C09078=1071.190,436.520,-116.526,176.537,35.842,156.699
C09079=1071.199,436.766,-116.574,176.544,35.855,156.702
C09080=1071.208,437.011,-116.622,176.552,35.868,156.705
C09081=1071.216,437.256,-116.669,176.561,35.881,156.709
C09082=1071.225,437.501,-116.716,176.568,35.894,156.712
C09083=1071.234,437.746,-116.764,176.576,35.908,156.716
C09084=1071.243,437.991,-116.811,176.585,35.921,156.719
C09085=1071.251,438.238,-116.859,176.593,35.934,156.722
C09086=1071.260,438.482,-116.906,176.600,35.947,156.726
C09087=1071.269,438.727,-116.954,176.609,35.961,156.729
C09088=1071.279,438.973,-117.001,176.617,35.974,156.733
C09089=1071.287,439.218,-117.049,176.626,35.988,156.736
C09090=1071.296,439.463,-117.097,176.633,36.001,156.739
C09091=1071.304,439.709,-117.145,176.641,36.015,156.743
C09092=1071.313,439.954,-117.193,176.650,36.029,156.747
C09093=1071.322,440.198,-117.241,176.658,36.042,156.750
C09094=1071.331,440.444,-117.289,176.667,36.056,156.754
C09095=1071.340,440.689,-117.337,176.675,36.069,156.757
C09096=1071.348,440.933,-117.385,176.684,36.083,156.761
C09097=1071.358,441.193,-117.437,176.693,36.098,156.764
C09098=1071.367,441.451,-117.487,176.702,36.113,156.768
C09099=1071.376,441.709,-117.538,176.711,36.127,156.772
C09100=1071.386,441.968,-117.589,176.720,36.142,156.776
C09101=1071.395,442.213,-117.637,176.728,36.156,156.779
C09102=1071.404,442.459,-117.686,176.737,36.170,156.783
C09103=1071.413,442.703,-117.734,176.745,36.184,156.787
C09104=1071.422,442.949,-117.782,176.754,36.199,156.791
C09105=1071.431,443.193,-117.831,176.763,36.213,156.794
C09106=1071.440,443.438,-117.880,176.771,36.227,156.798
C09107=1071.449,443.684,-117.929,176.780,36.241,156.802
C09108=1071.458,443.928,-117.977,176.789,36.256,156.805
C09109=1071.467,444.173,-118.026,176.798,36.270,156.809
C09110=1071.476,444.418,-118.075,176.806,36.285,156.813
C09111=1071.485,444.663,-118.123,176.816,36.299,156.817
C09112=1071.494,444.908,-118.172,176.825,36.314,156.821
C09113=1071.503,445.153,-118.222,176.834,36.329,156.824
C09114=1071.512,445.399,-118.271,176.842,36.343,156.828
C09115=1071.522,445.642,-118.320,176.851,36.358,156.832
C09116=1071.531,445.887,-118.369,176.861,36.373,156.836
C09117=1071.540,446.133,-118.418,176.870,36.388,156.840
C09118=1071.549,446.377,-118.468,176.879,36.402,156.844
C09119=1071.559,446.622,-118.516,176.888,36.417,156.848
C09120=1071.568,446.868,-118.565,176.898,36.433,156.852
C09121=1071.577,447.112,-118.615,176.907,36.447,156.856
C09122=1071.586,447.356,-118.665,176.916,36.463,156.860
C09123=1071.596,447.601,-118.713,176.926,36.477,156.864
C09124=1071.606,447.847,-118.763,176.934,36.493,156.868
C09125=1071.615,448.091,-118.813,176.943,36.508,156.872
C09126=1071.624,448.334,-118.862,176.952,36.523,156.876
C09127=1071.634,448.579,-118.911,176.959,36.538,156.880
C09128=1071.646,448.822,-118.959,176.967,36.552,156.883
C09129=1071.658,449.067,-119.006,176.976,36.566,156.887
C09130=1071.672,449.312,-119.053,176.983,36.579,156.891
C09131=1071.687,449.558,-119.100,176.990,36.592,156.894
C09132=1071.704,449.803,-119.144,176.997,36.604,156.897
C09133=1071.353,449.802,-119.394,176.982,36.746,156.935
C09134=1071.337,449.558,-119.348,176.975,36.734,156.932
C09135=1071.322,449.311,-119.302,176.968,36.722,156.929
C09136=1071.308,449.066,-119.255,176.960,36.708,156.925
C09137=1071.295,448.822,-119.208,176.953,36.695,156.921
C09138=1071.283,448.577,-119.160,176.944,36.680,156.918
C09139=1071.272,448.333,-119.111,176.936,36.666,156.914
C09140=1071.264,448.089,-119.062,176.927,36.650,156.910
C09141=1071.254,447.846,-119.012,176.918,36.636,156.906
C09142=1071.245,447.601,-118.962,176.908,36.620,156.902
C09143=1071.236,447.356,-118.913,176.899,36.605,156.898
C09144=1071.225,447.112,-118.864,176.890,36.590,156.894
C09145=1071.216,446.867,-118.814,176.880,36.575,156.890
C09146=1071.207,446.622,-118.765,176.871,36.560,156.886
C09147=1071.198,446.377,-118.715,176.862,36.545,156.882
C09148=1071.188,446.132,-118.667,176.853,36.531,156.878
C09149=1071.179,445.888,-118.617,176.844,36.516,156.874
C09150=1071.170,445.642,-118.568,176.834,36.501,156.870
C09151=1071.161,445.397,-118.519,176.825,36.486,156.866
C09152=1071.151,445.153,-118.470,176.816,36.472,156.862
C09153=1071.142,444.908,-118.421,176.806,36.457,156.858
C09154=1071.133,444.663,-118.371,176.798,36.443,156.855
C09155=1071.124,444.418,-118.322,176.789,36.428,156.851
C09156=1071.115,444.173,-118.274,176.780,36.413,156.847
C09157=1071.106,443.928,-118.225,176.771,36.399,156.843
C09158=1071.097,443.683,-118.176,176.762,36.385,156.839
C09159=1071.088,443.438,-118.128,176.753,36.370,156.836
C09160=1071.079,443.193,-118.079,176.744,36.356,156.832
C09161=1071.069,442.948,-118.030,176.735,36.342,156.828
C09162=1071.061,442.706,-117.982,176.727,36.328,156.825
C09163=1071.052,442.463,-117.933,176.718,36.314,156.821
C09164=1071.042,442.220,-117.885,176.710,36.300,156.817
C09165=1071.034,441.978,-117.838,176.701,36.286,156.814
C09166=1071.025,441.735,-117.790,176.693,36.272,156.810
C09167=1071.016,441.493,-117.742,176.684,36.259,156.806
C09168=1071.007,441.250,-117.694,176.676,36.245,156.803
C09169=1070.999,441.007,-117.647,176.667,36.231,156.799
C09170=1070.989,440.762,-117.598,176.659,36.217,156.796
C09171=1070.981,440.517,-117.550,176.650,36.203,156.792
C09172=1070.971,440.272,-117.502,176.642,36.190,156.789
C09173=1070.962,440.027,-117.454,176.633,36.176,156.785
C09174=1070.954,439.782,-117.406,176.625,36.163,156.782
C09175=1070.945,439.537,-117.358,176.616,36.149,156.778
C09176=1070.937,439.291,-117.310,176.608,36.135,156.774
C09177=1070.928,439.046,-117.263,176.599,36.122,156.771
C09178=1070.918,438.801,-117.215,176.591,36.108,156.768
C09179=1070.910,438.556,-117.167,176.584,36.095,156.764
C09180=1070.901,438.311,-117.120,176.575,36.082,156.761
C09181=1070.892,438.065,-117.072,176.567,36.068,156.757
C09182=1070.883,437.820,-117.024,176.559,36.055,156.754
C09183=1070.874,437.575,-116.977,176.550,36.042,156.750
C09184=1070.866,437.330,-116.929,176.543,36.029,156.747
C09185=1070.857,437.085,-116.881,176.535,36.016,156.744
C09186=1070.848,436.839,-116.834,176.526,36.003,156.741
C09187=1070.839,436.594,-116.787,176.518,35.990,156.737
C09188=1070.831,436.349,-116.740,176.511,35.977,156.734
C09189=1070.822,436.104,-116.693,176.502,35.964,156.731
C09190=1070.813,435.859,-116.645,176.494,35.951,156.727
C09191=1070.805,435.612,-116.597,176.486,35.938,156.724
C09192=1070.796,435.367,-116.550,176.479,35.925,156.721
C09193=1070.787,435.122,-116.503,176.471,35.912,156.717
C09194=1070.779,434.876,-116.457,176.463,35.900,156.714
C09195=1070.770,434.632,-116.409,176.455,35.887,156.711
C09196=1070.761,434.386,-116.362,176.447,35.874,156.708
C09197=1070.753,434.140,-116.316,176.440,35.862,156.705
C09198=1070.744,433.895,-116.269,176.432,35.849,156.701
C09199=1070.736,433.651,-116.222,176.424,35.837,156.698
C09200=1070.727,433.405,-116.175,176.417,35.824,156.695
C09201=1070.719,433.160,-116.128,176.409,35.811,156.692
C09202=1070.711,432.914,-116.081,176.402,35.799,156.689
C09203=1070.702,432.668,-116.034,176.394,35.787,156.686
C09204=1070.694,432.423,-115.988,176.387,35.774,156.683
C09205=1070.685,432.177,-115.941,176.379,35.762,156.679
C09206=1070.677,431.933,-115.895,176.372,35.750,156.676
C09207=1070.669,431.686,-115.849,176.364,35.738,156.673
C09208=1070.661,431.441,-115.802,176.357,35.725,156.670
C09209=1070.652,431.195,-115.755,176.349,35.713,156.667
C09210=1070.643,430.950,-115.709,176.342,35.701,156.664
C09211=1070.635,430.705,-115.663,176.334,35.689,156.661
C09212=1070.627,430.459,-115.617,176.327,35.677,156.658
C09213=1070.618,430.213,-115.571,176.320,35.665,156.655
C09214=1070.610,429.968,-115.524,176.312,35.653,156.652
C09215=1070.601,429.723,-115.479,176.305,35.641,156.649
C09216=1070.593,429.477,-115.432,176.297,35.629,156.646
C09217=1070.585,429.231,-115.386,176.290,35.617,156.643
C09218=1070.577,428.986,-115.340,176.283,35.606,156.640
C09219=1070.568,428.740,-115.294,176.276,35.594,156.637
C09220=1070.560,428.495,-115.249,176.269,35.582,156.634
C09221=1070.552,428.249,-115.202,176.262,35.570,156.632
C09222=1070.542,427.953,-115.146,176.253,35.556,156.628
C09223=1070.532,427.658,-115.091,176.244,35.542,156.625
C09224=1070.522,427.362,-115.037,176.236,35.528,156.621
C09225=1070.512,427.066,-114.982,176.227,35.514,156.618
C09226=1070.504,426.820,-114.936,176.220,35.503,156.615
C09227=1070.496,426.575,-114.891,176.214,35.492,156.612
C09228=1070.487,426.329,-114.845,176.207,35.480,156.609
C09229=1070.479,426.084,-114.800,176.199,35.469,156.607
C09230=1070.471,425.838,-114.754,176.192,35.457,156.604
C09231=1070.462,425.593,-114.709,176.186,35.446,156.601
C09232=1070.454,425.347,-114.663,176.179,35.435,156.598
C09233=1070.446,425.101,-114.619,176.171,35.423,156.595
C09234=1070.438,424.855,-114.573,176.165,35.412,156.593
C09235=1070.429,424.610,-114.528,176.158,35.401,156.590
C09236=1070.422,424.363,-114.483,176.151,35.390,156.587
C09237=1070.413,424.118,-114.437,176.145,35.379,156.584
C09238=1070.405,423.872,-114.392,176.138,35.368,156.582
C09239=1070.397,423.626,-114.347,176.131,35.357,156.579
C09240=1070.389,423.381,-114.302,176.124,35.346,156.576
C09241=1070.381,423.135,-114.257,176.117,35.335,156.574
C09242=1070.373,422.889,-114.212,176.111,35.324,156.571
C09243=1070.365,422.643,-114.167,176.104,35.313,156.568
C09244=1070.357,422.398,-114.123,176.098,35.302,156.566
C09245=1070.349,422.152,-114.077,176.091,35.291,156.563
C09246=1070.341,421.906,-114.032,176.085,35.280,156.560
C09247=1070.333,421.660,-113.988,176.077,35.269,156.558
C09248=1070.325,421.415,-113.942,176.071,35.259,156.555
C09249=1070.317,421.169,-113.898,176.064,35.248,156.552
C09250=1070.309,420.923,-113.854,176.058,35.237,156.550
C09251=1070.301,420.676,-113.808,176.051,35.227,156.547
C09252=1070.293,420.431,-113.764,176.045,35.216,156.545
C09253=1070.285,420.185,-113.720,176.039,35.205,156.542
C09254=1070.277,419.939,-113.675,176.032,35.195,156.540
C09255=1070.269,419.693,-113.631,176.026,35.184,156.537
C09256=1070.262,419.447,-113.586,176.019,35.174,156.534
C09257=1070.254,419.202,-113.542,176.013,35.164,156.532
C09258=1070.246,418.955,-113.498,176.006,35.153,156.529
C09259=1070.238,418.709,-113.454,176.000,35.143,156.527
C09260=1070.230,418.464,-113.409,175.994,35.132,156.525
C09261=1070.222,418.218,-113.365,175.987,35.122,156.522
C09262=1070.214,417.972,-113.321,175.981,35.112,156.520
C09263=1070.206,417.726,-113.277,175.975,35.101,156.517
C09264=1070.198,417.480,-113.232,175.968,35.091,156.515
C09265=1070.191,417.233,-113.189,175.962,35.081,156.512
C09266=1070.183,416.988,-113.144,175.956,35.071,156.510
C09267=1070.175,416.742,-113.100,175.950,35.061,156.507
C09268=1070.167,416.496,-113.056,175.944,35.050,156.505
C09269=1070.159,416.250,-113.012,175.938,35.040,156.502
C09270=1070.151,416.004,-112.968,175.932,35.030,156.500
C09271=1070.143,415.757,-112.925,175.925,35.020,156.498
C09272=1070.136,415.512,-112.881,175.919,35.010,156.495
C09273=1070.128,415.266,-112.837,175.913,35.000,156.493
C09274=1070.120,415.020,-112.793,175.907,34.990,156.490
C09275=1070.112,414.774,-112.749,175.901,34.980,156.488
C09276=1070.104,414.527,-112.706,175.894,34.970,156.486
C09277=1070.097,414.281,-112.662,175.889,34.960,156.483
C09278=1070.088,414.004,-112.613,175.882,34.949,156.481
C09279=1070.079,413.728,-112.564,175.875,34.938,156.478
C09280=1070.071,413.451,-112.515,175.869,34.927,156.475
C09281=1070.061,413.174,-112.466,175.862,34.916,156.473
C09282=1070.050,412.806,-112.402,175.853,34.902,156.469
C09283=1070.039,412.438,-112.336,175.843,34.887,156.466
C09284=1070.027,412.069,-112.272,175.835,34.873,156.463
C09285=1070.015,411.700,-112.207,175.826,34.859,156.459
C09286=1070.007,411.454,-112.164,175.820,34.849,156.457
C09287=1070.000,411.208,-112.121,175.815,34.840,156.455
C09288=1069.992,410.962,-112.077,175.809,34.830,156.452
C09289=1069.984,410.715,-112.035,175.803,34.821,156.450
C09290=1069.977,410.470,-111.991,175.797,34.811,156.448
C09291=1069.969,410.224,-111.948,175.791,34.802,156.446
C09292=1069.962,409.977,-111.906,175.786,34.793,156.444
C09293=1069.954,409.731,-111.862,175.780,34.783,156.441
C09294=1069.946,409.485,-111.820,175.774,34.774,156.439
C09295=1069.939,409.239,-111.777,175.769,34.764,156.437
C09296=1069.932,408.993,-111.733,175.763,34.755,156.435
C09297=1069.923,408.746,-111.691,175.757,34.746,156.433
C09298=1069.916,408.501,-111.648,175.751,34.737,156.431
C09299=1069.909,408.254,-111.605,175.746,34.727,156.428
C09300=1069.901,408.008,-111.563,175.740,34.718,156.426
C09301=1069.894,407.762,-111.520,175.734,34.709,156.424
C09302=1069.887,407.515,-111.477,175.729,34.700,156.422
C09303=1069.879,407.269,-111.435,175.723,34.690,156.420
C09304=1069.871,407.023,-111.391,175.717,34.681,156.418
C09305=1069.864,406.776,-111.349,175.712,34.672,156.416
C09306=1069.857,406.530,-111.307,175.707,34.663,156.413
C09307=1069.849,406.283,-111.264,175.701,34.654,156.411
C09308=1069.842,406.038,-111.222,175.696,34.645,156.409
C09309=1069.835,405.792,-111.179,175.690,34.636,156.407
C09310=1069.826,405.545,-111.136,175.684,34.627,156.405
C09311=1069.819,405.299,-111.094,175.679,34.618,156.403
C09312=1069.812,405.053,-111.052,175.673,34.609,156.401
C09313=1069.804,404.807,-111.010,175.667,34.600,156.399
C09314=1069.797,404.560,-110.967,175.663,34.592,156.397
C09315=1069.789,404.314,-110.925,175.657,34.583,156.395
C09316=1069.782,404.068,-110.882,175.651,34.574,156.393
C09317=1069.775,403.821,-110.841,175.646,34.565,156.391
C09318=1069.767,403.574,-110.799,175.640,34.557,156.389
C09319=1069.760,403.328,-110.756,175.636,34.548,156.387
C09320=1069.752,403.082,-110.714,175.630,34.539,156.385
C09321=1069.745,402.836,-110.672,175.624,34.530,156.383
C09322=1069.738,402.590,-110.631,175.619,34.522,156.381
C09323=1069.731,402.343,-110.589,175.613,34.513,156.379
C09324=1069.723,402.097,-110.546,175.609,34.505,156.377
C09325=1069.715,401.850,-110.505,175.603,34.496,156.375
C09326=1069.708,401.604,-110.463,175.598,34.487,156.373
C09327=1069.700,401.358,-110.421,175.592,34.479,156.371
C09328=1069.693,401.111,-110.379,175.587,34.470,156.369
C09329=1069.686,400.865,-110.338,175.582,34.462,156.367
C09330=1069.674,400.468,-110.271,175.573,34.448,156.364
C09331=1069.662,400.071,-110.203,175.565,34.434,156.361
C09332=1069.650,399.674,-110.137,175.556,34.421,156.358
C09333=1069.639,399.277,-110.069,175.548,34.408,156.354
C09334=1069.631,399.031,-110.028,175.543,34.399,156.353
C09335=1069.624,398.784,-109.987,175.537,34.391,156.351
C09336=1069.616,398.538,-109.945,175.533,34.383,156.349
C09337=1069.609,398.291,-109.904,175.527,34.374,156.347
C09338=1069.602,398.045,-109.862,175.523,34.366,156.345
C09339=1069.595,397.798,-109.821,175.517,34.358,156.343
C09340=1069.587,397.552,-109.780,175.512,34.350,156.341
C09341=1069.580,397.306,-109.738,175.507,34.341,156.339
C09342=1069.572,397.059,-109.697,175.502,34.333,156.337
C09343=1069.566,396.813,-109.656,175.497,34.325,156.336
C09344=1069.558,396.567,-109.615,175.492,34.317,156.334
C09345=1069.551,396.320,-109.573,175.487,34.309,156.332
C09346=1069.544,396.073,-109.532,175.482,34.301,156.330
C09347=1069.537,395.827,-109.491,175.477,34.293,156.328
C09348=1069.529,395.580,-109.450,175.471,34.284,156.326
C09349=1069.523,395.334,-109.409,175.467,34.277,156.325
C09350=1069.515,395.088,-109.368,175.461,34.268,156.323
C09351=1069.508,394.841,-109.328,175.457,34.261,156.321
C09352=1069.500,394.594,-109.287,175.451,34.253,156.319
C09353=1069.494,394.348,-109.246,175.447,34.245,156.317
C09354=1069.486,394.102,-109.204,175.441,34.237,156.316
C09355=1069.479,393.855,-109.163,175.437,34.229,156.314
C09356=1069.473,393.609,-109.123,175.432,34.221,156.312
C09357=1069.465,393.362,-109.082,175.426,34.213,156.310
C09358=1069.457,393.116,-109.041,175.422,34.205,156.309
C09359=1069.451,392.869,-109.001,175.416,34.197,156.307
C09360=1069.443,392.623,-108.960,175.412,34.190,156.305
C09361=1069.436,392.376,-108.919,175.406,34.182,156.303
C09362=1069.429,392.130,-108.879,175.402,34.174,156.302
C09363=1069.422,391.883,-108.838,175.397,34.166,156.300
C09364=1069.414,391.636,-108.798,175.392,34.159,156.298
C09365=1069.408,391.390,-108.757,175.387,34.151,156.296
C09366=1069.401,391.143,-108.716,175.382,34.143,156.295
C09367=1069.393,390.898,-108.676,175.377,34.136,156.293
C09368=1069.386,390.650,-108.636,175.373,34.128,156.291
C09369=1069.379,390.405,-108.595,175.367,34.120,156.289
C09370=1069.372,390.158,-108.555,175.363,34.113,156.288
C09371=1069.364,389.911,-108.515,175.359,34.105,156.286
C09372=1069.357,389.665,-108.474,175.353,34.098,156.285
C09373=1069.350,389.418,-108.434,175.349,34.090,156.283
C09374=1069.343,389.171,-108.394,175.343,34.083,156.281
C09375=1069.336,388.925,-108.354,175.339,34.075,156.279
C09376=1069.329,388.678,-108.314,175.334,34.068,156.278
C09377=1069.321,388.432,-108.273,175.329,34.061,156.276
C09378=1069.314,388.186,-108.234,175.324,34.053,156.274
C09379=1069.307,387.938,-108.193,175.320,34.045,156.273
C09380=1069.300,387.692,-108.154,175.315,34.038,156.271
C09381=1069.293,387.445,-108.113,175.310,34.030,156.269
C09382=1069.286,387.199,-108.074,175.306,34.023,156.268
C09383=1069.279,386.952,-108.034,175.300,34.016,156.266
C09384=1069.272,386.705,-107.994,175.296,34.009,156.265
C09385=1069.265,386.459,-107.954,175.292,34.001,156.263
C09386=1069.257,386.202,-107.912,175.286,33.993,156.261
C09387=1069.250,385.945,-107.871,175.282,33.986,156.260
C09388=1069.243,385.688,-107.829,175.277,33.978,156.258
C09389=1069.235,385.431,-107.787,175.271,33.970,156.256
C09390=1069.229,385.184,-107.747,175.267,33.964,156.255
C09391=1069.222,384.937,-107.708,175.263,33.956,156.253
C09392=1069.214,384.690,-107.668,175.257,33.949,156.252
C09393=1069.208,384.444,-107.628,175.253,33.942,156.250
C09394=1069.200,384.198,-107.589,175.249,33.935,156.248
C09395=1069.194,383.951,-107.550,175.243,33.927,156.247
C09396=1069.187,383.704,-107.509,175.239,33.920,156.245
C09397=1069.180,383.457,-107.470,175.235,33.913,156.244
C09398=1069.173,383.210,-107.431,175.231,33.906,156.242
C09399=1069.166,382.964,-107.391,175.225,33.899,156.240
C09400=1069.159,382.717,-107.351,175.221,33.892,156.239
C09401=1069.152,382.470,-107.312,175.217,33.885,156.237
C09402=1069.145,382.224,-107.272,175.211,33.877,156.236
C09403=1069.139,381.977,-107.233,175.207,33.870,156.234
C09404=1069.132,381.731,-107.194,175.203,33.863,156.233
C09405=1069.125,381.484,-107.154,175.199,33.856,156.231
C09406=1069.118,381.237,-107.114,175.193,33.849,156.230
C09407=1069.111,380.990,-107.075,175.189,33.842,156.228
C09408=1069.104,380.744,-107.036,175.185,33.836,156.227
C09409=1069.097,380.497,-106.997,175.180,33.828,156.225
C09410=1069.090,380.249,-106.958,175.175,33.821,156.224
C09411=1069.083,380.002,-106.919,175.171,33.815,156.222
C09412=1069.076,379.756,-106.879,175.167,33.808,156.221
C09413=1069.069,379.509,-106.841,175.162,33.801,156.219
C09414=1069.062,379.263,-106.802,175.157,33.794,156.218
C09415=1069.055,379.016,-106.763,175.153,33.787,156.216
C09416=1069.048,378.770,-106.723,175.149,33.780,156.215
C09417=1069.041,378.523,-106.684,175.144,33.773,156.213
C09418=1069.034,378.276,-106.646,175.140,33.767,156.212
C09419=1069.027,378.028,-106.606,175.135,33.760,156.210
C09420=1069.020,377.782,-106.568,175.131,33.753,156.209
C09421=1069.013,377.535,-106.529,175.126,33.746,156.207
C09422=1069.007,377.288,-106.490,175.122,33.740,156.206
C09423=1069.000,377.041,-106.451,175.118,33.733,156.204
C09424=1068.993,376.794,-106.412,175.113,33.726,156.203
C09425=1068.986,376.547,-106.373,175.109,33.720,156.201
C09426=1068.979,376.301,-106.335,175.104,33.713,156.200
C09427=1068.973,376.054,-106.296,175.100,33.706,156.199
C09428=1068.966,375.807,-106.257,175.096,33.700,156.197
C09429=1068.959,375.560,-106.218,175.092,33.693,156.196
C09430=1068.951,375.314,-106.180,175.087,33.686,156.194
C09431=1068.945,375.068,-106.141,175.082,33.679,156.193
C09432=1068.939,374.820,-106.103,175.078,33.673,156.191
C09433=1068.932,374.573,-106.064,175.074,33.666,156.190
C09434=1068.925,374.326,-106.026,175.070,33.659,156.188
C09435=1068.918,374.080,-105.987,175.065,33.653,156.187
C09436=1068.911,373.833,-105.948,175.061,33.646,156.186
C09437=1068.905,373.585,-105.910,175.057,33.640,156.184
C09438=1068.898,373.349,-105.873,175.053,33.634,156.183
C09439=1068.892,373.112,-105.836,175.049,33.628,156.182
C09440=1068.886,372.875,-105.799,175.045,33.621,156.180
C09441=1068.879,372.638,-105.762,175.040,33.615,156.179
C09442=1068.872,372.401,-105.726,175.036,33.609,156.178
C09443=1068.866,372.164,-105.689,175.032,33.602,156.176
C09444=1068.859,371.927,-105.652,175.028,33.596,156.175
C09445=1068.852,371.689,-105.615,175.024,33.590,156.174
C09446=1068.845,371.443,-105.577,175.019,33.584,156.172
C09447=1068.839,371.196,-105.539,175.015,33.577,156.171
C09448=1068.832,370.949,-105.501,175.011,33.571,156.170
C09449=1068.825,370.702,-105.463,175.007,33.565,156.168
C09450=1068.818,370.455,-105.425,175.003,33.559,156.167
C09451=1068.812,370.208,-105.386,174.999,33.552,156.166
C09452=1068.805,369.961,-105.349,174.994,33.546,156.164
C09453=1068.798,369.714,-105.311,174.990,33.540,156.163
C09454=1068.791,369.467,-105.272,174.986,33.533,156.162
C09455=1068.784,369.220,-105.234,174.982,33.527,156.160
C09456=1068.778,368.973,-105.197,174.978,33.521,156.159
C09457=1068.771,368.726,-105.159,174.974,33.514,156.158
C09458=1068.764,368.479,-105.120,174.969,33.508,156.156
C09459=1068.758,368.233,-105.083,174.965,33.502,156.155
C09460=1068.751,367.985,-105.045,174.960,33.495,156.154
C09461=1068.744,367.738,-105.007,174.956,33.489,156.152
C09462=1068.737,367.491,-104.969,174.952,33.483,156.151
C09463=1068.731,367.244,-104.932,174.948,33.477,156.150
C09464=1068.724,366.997,-104.894,174.944,33.471,156.148
C09465=1068.718,366.750,-104.857,174.940,33.465,156.147
C09466=1068.711,366.503,-104.819,174.936,33.458,156.146
C09467=1068.704,366.256,-104.781,174.932,33.452,156.144
C09468=1068.698,366.009,-104.743,174.928,33.446,156.143
C09469=1068.692,365.762,-104.705,174.924,33.440,156.142
C09470=1068.684,365.515,-104.668,174.920,33.434,156.140
C09471=1068.678,365.268,-104.630,174.916,33.428,156.139
C09472=1068.671,365.021,-104.593,174.912,33.422,156.138
C09473=1068.665,364.774,-104.555,174.907,33.415,156.137
C09474=1068.658,364.527,-104.517,174.903,33.409,156.135
C09475=1068.651,364.280,-104.480,174.899,33.403,156.134
C09476=1068.645,364.033,-104.442,174.895,33.397,156.133
C09477=1068.638,363.785,-104.405,174.891,33.391,156.132
C09478=1068.631,363.539,-104.368,174.887,33.385,156.130
C09479=1068.625,363.291,-104.330,174.883,33.379,156.129
C09480=1068.618,363.044,-104.293,174.879,33.373,156.128
C09481=1068.611,362.797,-104.256,174.874,33.367,156.127
C09482=1068.605,362.551,-104.219,174.870,33.362,156.125
C09483=1068.598,362.303,-104.181,174.866,33.355,156.124
C09484=1068.592,362.056,-104.144,174.862,33.349,156.123
C09485=1068.584,361.809,-104.107,174.859,33.344,156.122
C09486=1068.578,361.561,-104.070,174.855,33.337,156.120
C09487=1068.571,361.315,-104.033,174.851,33.332,156.119
C09488=1068.565,361.067,-103.996,174.847,33.326,156.118
C09489=1068.558,360.820,-103.958,174.843,33.320,156.117
C09490=1068.552,360.573,-103.922,174.838,33.314,156.115
C09491=1068.544,360.326,-103.884,174.834,33.308,156.114
C09492=1068.538,360.079,-103.848,174.830,33.302,156.113
C09493=1068.532,359.832,-103.810,174.826,33.296,156.112
C09494=1068.526,359.604,-103.776,174.823,33.291,156.111
C09495=1068.520,359.375,-103.741,174.819,33.286,156.110
C09496=1068.514,359.147,-103.707,174.816,33.280,156.108
C09497=1068.507,358.918,-103.673,174.812,33.275,156.107
C09498=1068.501,358.690,-103.639,174.809,33.270,156.106
C09499=1068.495,358.462,-103.605,174.805,33.264,156.105
C09500=1068.489,358.233,-103.572,174.801,33.259,156.104
C09501=1068.483,358.004,-103.537,174.798,33.253,156.103
C09502=1068.476,357.757,-103.501,174.793,33.248,156.102
C09503=1068.470,357.510,-103.464,174.789,33.242,156.101
C09504=1068.463,357.263,-103.427,174.785,33.237,156.099
C09505=1068.457,357.016,-103.390,174.781,33.231,156.098
C09506=1068.450,356.768,-103.354,174.778,33.225,156.097
C09507=1068.443,356.521,-103.317,174.774,33.219,156.096
C09508=1068.437,356.274,-103.280,174.770,33.214,156.095
C09509=1068.430,356.027,-103.243,174.766,33.208,156.093
C09510=1068.423,355.780,-103.207,174.762,33.202,156.092
C09511=1068.417,355.533,-103.170,174.759,33.197,156.091
C09512=1068.411,355.285,-103.134,174.755,33.191,156.090
C09513=1068.404,355.038,-103.097,174.751,33.185,156.089
C09514=1068.397,354.791,-103.061,174.747,33.180,156.088
C09515=1068.391,354.544,-103.024,174.743,33.174,156.087
C09516=1068.384,354.296,-102.987,174.740,33.169,156.085
C09517=1068.377,354.049,-102.951,174.735,33.163,156.084
C09518=1068.371,353.802,-102.915,174.731,33.157,156.083
C09519=1068.365,353.554,-102.879,174.727,33.152,156.082
C09520=1068.358,353.307,-102.843,174.723,33.146,156.081
C09521=1068.351,353.060,-102.806,174.720,33.141,156.080
C09522=1068.345,352.812,-102.770,174.716,33.135,156.078
C09523=1068.339,352.565,-102.733,174.712,33.129,156.077
C09524=1068.332,352.318,-102.697,174.708,33.124,156.076
C09525=1068.326,352.071,-102.661,174.705,33.118,156.075
C09526=1068.319,351.823,-102.625,174.701,33.113,156.074
C09527=1068.312,351.576,-102.588,174.697,33.107,156.073
C09528=1068.306,351.329,-102.552,174.693,33.102,156.072
C09529=1068.300,351.081,-102.516,174.690,33.096,156.071
C09530=1068.293,350.835,-102.480,174.686,33.091,156.069
C09531=1068.286,350.587,-102.443,174.682,33.086,156.068
C09532=1068.280,350.339,-102.408,174.678,33.080,156.067
C09533=1068.273,350.093,-102.372,174.675,33.075,156.066
C09534=1068.267,349.845,-102.336,174.671,33.069,156.065
C09535=1068.261,349.598,-102.300,174.667,33.063,156.064
C09536=1068.254,349.350,-102.264,174.664,33.058,156.063
C09537=1068.247,349.103,-102.228,174.660,33.053,156.062
C09538=1068.241,348.856,-102.192,174.656,33.048,156.061
C09539=1068.234,348.608,-102.156,174.651,33.042,156.059
C09540=1068.228,348.361,-102.120,174.648,33.036,156.058
C09541=1068.221,348.114,-102.084,174.644,33.031,156.057
C09542=1068.215,347.866,-102.048,174.640,33.026,156.056
C09543=1068.208,347.619,-102.012,174.637,33.021,156.055
C09544=1068.202,347.371,-101.977,174.633,33.015,156.054
C09545=1068.195,347.124,-101.942,174.629,33.010,156.053
C09546=1068.189,346.877,-101.905,174.626,33.004,156.052
C09547=1068.183,346.629,-101.869,174.622,32.999,156.051
C09548=1068.176,346.382,-101.834,174.618,32.994,156.050
C09549=1068.170,346.135,-101.798,174.615,32.988,156.049
C09550=1068.163,345.908,-101.765,174.611,32.984,156.048
C09551=1068.158,345.682,-101.733,174.608,32.979,156.047
C09552=1068.153,345.455,-101.700,174.605,32.974,156.046
C09553=1068.146,345.229,-101.667,174.601,32.969,156.045
C09554=1068.141,345.003,-101.635,174.598,32.964,156.044
C09555=1068.134,344.776,-101.602,174.595,32.959,156.043
C09556=1068.129,344.549,-101.569,174.591,32.955,156.042
C09557=1068.123,344.323,-101.537,174.588,32.949,156.041
C09558=1068.117,344.076,-101.502,174.584,32.945,156.040
C09559=1068.110,343.828,-101.467,174.581,32.939,156.039
C09560=1068.104,343.581,-101.431,174.577,32.934,156.038
C09561=1068.097,343.333,-101.396,174.573,32.929,156.037
C09562=1068.091,343.086,-101.361,174.570,32.924,156.036
C09563=1068.084,342.838,-101.325,174.566,32.918,156.035
C09564=1068.078,342.591,-101.290,174.562,32.913,156.034
C09565=1068.071,342.344,-101.255,174.559,32.908,156.033
C09566=1068.065,342.096,-101.219,174.555,32.903,156.031
C09567=1068.058,341.849,-101.184,174.552,32.898,156.031
C09568=1068.051,341.601,-101.149,174.548,32.893,156.029
C09569=1068.045,341.354,-101.113,174.544,32.887,156.028
C09570=1068.039,341.106,-101.079,174.541,32.882,156.027
C09571=1068.033,340.859,-101.044,174.537,32.877,156.026
C09572=1068.027,340.611,-101.008,174.534,32.872,156.025
C09573=1068.020,340.364,-100.973,174.530,32.867,156.024
C09574=1068.013,340.116,-100.938,174.527,32.862,156.023
C09575=1068.007,339.869,-100.902,174.523,32.857,156.022
C09576=1068.001,339.621,-100.868,174.519,32.852,156.021
C09577=1067.994,339.374,-100.833,174.516,32.847,156.020
C09578=1067.988,339.127,-100.798,174.512,32.841,156.019
C09579=1067.982,338.879,-100.762,174.509,32.837,156.018
C09580=1067.975,338.631,-100.728,174.505,32.831,156.017
C09581=1067.969,338.384,-100.693,174.502,32.827,156.016
C09582=1067.962,338.137,-100.658,174.498,32.821,156.015
C09583=1067.957,337.889,-100.623,174.494,32.816,156.014
C09584=1067.950,337.641,-100.587,174.491,32.811,156.013
C09585=1067.944,337.394,-100.553,174.487,32.806,156.012
C09586=1067.937,337.147,-100.518,174.484,32.801,156.011
C09587=1067.930,336.899,-100.483,174.480,32.796,156.010
C09588=1067.924,336.651,-100.449,174.477,32.791,156.009
C09589=1067.918,336.405,-100.414,174.473,32.786,156.008
C09590=1067.912,336.156,-100.379,174.470,32.781,156.007
C09591=1067.905,335.909,-100.344,174.466,32.776,156.006
C09592=1067.899,335.661,-100.309,174.463,32.771,156.005
C09593=1067.893,335.414,-100.275,174.459,32.766,156.004
C09594=1067.886,335.166,-100.240,174.456,32.761,156.003
C09595=1067.880,334.918,-100.206,174.453,32.756,156.002
C09596=1067.874,334.672,-100.171,174.450,32.752,156.001
C09597=1067.867,334.424,-100.137,174.446,32.746,156.000
C09598=1067.861,334.176,-100.102,174.443,32.742,155.999
C09599=1067.854,333.929,-100.067,174.439,32.737,155.998
C09600=1067.848,333.681,-100.033,174.436,32.732,155.997
C09601=1067.842,333.433,-99.999,174.432,32.727,155.996
C09602=1067.835,333.187,-99.964,174.429,32.722,155.996
C09603=1067.829,332.939,-99.929,174.425,32.717,155.995
C09604=1067.822,332.691,-99.895,174.422,32.712,155.994
C09605=1067.817,332.443,-99.861,174.418,32.707,155.993
C09606=1067.811,332.214,-99.829,174.415,32.703,155.992
C09607=1067.805,331.986,-99.797,174.412,32.698,155.991
C09608=1067.799,331.757,-99.765,174.409,32.693,155.990
C09609=1067.793,331.527,-99.733,174.405,32.689,155.989
C09610=1067.787,331.299,-99.702,174.402,32.684,155.988
C09611=1067.781,331.069,-99.670,174.399,32.680,155.987
C09612=1067.775,330.840,-99.638,174.396,32.675,155.986
C09613=1067.770,330.612,-99.607,174.393,32.671,155.986
C09614=1067.763,330.364,-99.573,174.389,32.666,155.985
C09615=1067.757,330.117,-99.539,174.386,32.662,155.984
C09616=1067.750,329.869,-99.504,174.382,32.657,155.983
C09617=1067.743,329.621,-99.470,174.379,32.652,155.982
C09618=1067.737,329.374,-99.436,174.375,32.647,155.981
C09619=1067.731,329.126,-99.402,174.372,32.643,155.980
C09620=1067.724,328.879,-99.369,174.369,32.638,155.979
C09621=1067.718,328.631,-99.334,174.366,32.633,155.978
C09622=1067.712,328.383,-99.300,174.363,32.629,155.977
C09623=1067.705,328.136,-99.266,174.359,32.624,155.976
C09624=1067.698,327.887,-99.233,174.356,32.619,155.975
C09625=1067.692,327.640,-99.199,174.352,32.614,155.974
C09626=1067.685,327.392,-99.165,174.349,32.610,155.974
C09627=1067.680,327.145,-99.131,174.346,32.605,155.973
C09628=1067.672,326.897,-99.097,174.342,32.600,155.972
C09629=1067.666,326.650,-99.063,174.339,32.596,155.971
C09630=1067.660,326.402,-99.030,174.335,32.591,155.970
C09631=1067.654,326.154,-98.996,174.332,32.586,155.969
C09632=1067.647,325.907,-98.962,174.329,32.581,155.968
C09633=1067.641,325.659,-98.928,174.325,32.577,155.967
C09634=1067.635,325.412,-98.894,174.322,32.572,155.966
C09635=1067.628,325.164,-98.861,174.318,32.567,155.965
C09636=1067.622,324.917,-98.826,174.315,32.563,155.964
C09637=1067.615,324.668,-98.793,174.312,32.558,155.964
C09638=1067.609,324.421,-98.759,174.308,32.554,155.963
C09639=1067.603,324.174,-98.726,174.306,32.549,155.962
C09640=1067.597,323.925,-98.692,174.303,32.544,155.961
C09641=1067.591,323.678,-98.658,174.299,32.539,155.960
C09642=1067.584,323.430,-98.625,174.296,32.535,155.959
C09643=1067.578,323.183,-98.591,174.292,32.530,155.958
C09644=1067.572,322.935,-98.558,174.289,32.525,155.957
C09645=1067.565,322.687,-98.524,174.286,32.521,155.956
C09646=1067.559,322.439,-98.491,174.282,32.516,155.956
C09647=1067.553,322.192,-98.457,174.279,32.512,155.955
C09648=1067.546,321.944,-98.424,174.276,32.507,155.954
C09649=1067.540,321.697,-98.390,174.272,32.502,155.953
C09650=1067.534,321.449,-98.357,174.269,32.498,155.952
C09651=1067.528,321.202,-98.323,174.266,32.493,155.951
C09652=1067.521,320.953,-98.290,174.262,32.489,155.950
C09653=1067.515,320.706,-98.256,174.260,32.484,155.949
C09654=1067.509,320.459,-98.223,174.257,32.479,155.948
C09655=1067.503,320.211,-98.190,174.254,32.475,155.948
C09656=1067.496,319.963,-98.156,174.250,32.470,155.947
C09657=1067.491,319.715,-98.123,174.247,32.465,155.946
C09658=1067.484,319.467,-98.090,174.244,32.461,155.945
C09659=1067.479,319.220,-98.056,174.240,32.456,155.944
C09660=1067.472,318.972,-98.023,174.237,32.451,155.943
C09661=1067.465,318.724,-97.990,174.234,32.447,155.942
C09662=1067.460,318.492,-97.958,174.231,32.443,155.941
C09663=1067.454,318.260,-97.928,174.228,32.438,155.940
C09664=1067.448,318.028,-97.896,174.224,32.434,155.940
C09665=1067.443,317.796,-97.865,174.221,32.430,155.939
C09666=1067.437,317.564,-97.834,174.219,32.425,155.938
C09667=1067.431,317.332,-97.802,174.216,32.421,155.937
C09668=1067.426,317.101,-97.772,174.213,32.417,155.936
C09669=1067.420,316.869,-97.741,174.210,32.413,155.936
C09670=1067.414,316.621,-97.708,174.207,32.408,155.935
C09671=1067.407,316.373,-97.675,174.204,32.404,155.934
C09672=1067.402,316.125,-97.641,174.200,32.399,155.933
C09673=1067.395,315.877,-97.609,174.197,32.394,155.932
C09674=1067.390,315.630,-97.575,174.194,32.390,155.931
C09675=1067.384,315.382,-97.543,174.191,32.385,155.930
C09676=1067.377,315.134,-97.510,174.187,32.381,155.929
C09677=1067.372,314.886,-97.476,174.184,32.376,155.929
C09678=1067.365,314.639,-97.444,174.182,32.372,155.928
C09679=1067.359,314.391,-97.411,174.179,32.367,155.927
C09680=1067.354,314.143,-97.378,174.176,32.363,155.926
C09681=1067.347,313.896,-97.345,174.172,32.358,155.925
C09682=1067.341,313.648,-97.312,174.169,32.353,155.924
C09683=1067.334,313.400,-97.279,174.166,32.349,155.923
C09684=1067.328,313.152,-97.246,174.162,32.345,155.923
C09685=1067.322,312.905,-97.214,174.159,32.341,155.922
C09686=1067.315,312.657,-97.182,174.156,32.336,155.921
C09687=1067.309,312.409,-97.149,174.153,32.332,155.920
C09688=1067.302,312.162,-97.117,174.150,32.327,155.919
C09689=1067.296,311.914,-97.084,174.147,32.323,155.918
C09690=1067.290,311.666,-97.052,174.144,32.319,155.918
C09691=1067.284,311.418,-97.019,174.141,32.314,155.917
C09692=1067.277,311.171,-96.986,174.138,32.310,155.916
C09693=1067.271,310.923,-96.954,174.134,32.305,155.915
C09694=1067.264,310.674,-96.921,174.131,32.301,155.914
C09695=1067.258,310.426,-96.888,174.128,32.297,155.914
C09696=1067.251,310.179,-96.856,174.125,32.293,155.913
C09697=1067.245,309.931,-96.824,174.121,32.288,155.912
C09698=1067.239,309.683,-96.792,174.119,32.283,155.911
C09699=1067.233,309.436,-96.759,174.116,32.279,155.910
C09700=1067.227,309.188,-96.727,174.113,32.275,155.909
C09701=1067.221,308.941,-96.694,174.110,32.271,155.909
C09702=1067.215,308.692,-96.662,174.106,32.266,155.908
C09703=1067.208,308.445,-96.630,174.103,32.262,155.907
C09704=1067.202,308.198,-96.597,174.100,32.257,155.906
C09705=1067.196,307.949,-96.565,174.097,32.253,155.905
C09706=1067.189,307.702,-96.533,174.094,32.249,155.904
C09707=1067.183,307.454,-96.501,174.090,32.244,155.904
C09708=1067.177,307.206,-96.468,174.088,32.240,155.903
C09709=1067.170,306.958,-96.437,174.085,32.236,155.902
C09710=1067.164,306.711,-96.404,174.082,32.232,155.901
C09711=1067.158,306.462,-96.372,174.079,32.227,155.900
C09712=1067.152,306.214,-96.340,174.076,32.223,155.900
C09713=1067.146,305.967,-96.307,174.072,32.218,155.899
C09714=1067.140,305.719,-96.276,174.069,32.214,155.898
C09715=1067.133,305.472,-96.243,174.066,32.210,155.897
C09716=1067.127,305.223,-96.211,174.063,32.205,155.896
C09717=1067.121,304.975,-96.179,174.061,32.201,155.896
C09718=1067.115,304.746,-96.149,174.058,32.197,155.895
C09719=1067.110,304.516,-96.119,174.055,32.193,155.894
C09720=1067.104,304.285,-96.090,174.052,32.189,155.893
C09721=1067.098,304.055,-96.059,174.049,32.185,155.893
C09722=1067.093,303.824,-96.030,174.046,32.181,155.892
C09723=1067.087,303.594,-96.000,174.043,32.177,155.891
C09724=1067.081,303.364,-95.971,174.040,32.173,155.890
C09725=1067.076,303.134,-95.941,174.037,32.169,155.889
C09726=1067.070,302.886,-95.909,174.035,32.165,155.889
C09727=1067.064,302.638,-95.877,174.032,32.160,155.888
C09728=1067.057,302.391,-95.845,174.029,32.156,155.887
C09729=1067.051,302.143,-95.813,174.026,32.152,155.886
C09730=1067.045,301.895,-95.781,174.023,32.147,155.885
C09731=1067.039,301.647,-95.749,174.020,32.143,155.885
C09732=1067.033,301.399,-95.718,174.017,32.139,155.884
C09733=1067.027,301.151,-95.686,174.014,32.135,155.883
C09734=1067.021,300.903,-95.654,174.012,32.130,155.882
C09735=1067.016,300.655,-95.623,174.008,32.126,155.881
C09736=1067.009,300.408,-95.590,174.005,32.122,155.881
C09737=1067.003,300.160,-95.558,174.002,32.117,155.880
C09738=1066.997,299.912,-95.527,173.999,32.113,155.879
C09739=1066.991,299.665,-95.495,173.996,32.109,155.878
C09740=1066.985,299.416,-95.463,173.993,32.104,155.877
C09741=1066.979,299.169,-95.432,173.990,32.100,155.877
C09742=1066.973,298.921,-95.400,173.988,32.096,155.876
C09743=1066.967,298.673,-95.368,173.985,32.091,155.875
C09744=1066.961,298.425,-95.336,173.982,32.087,155.874
C09745=1066.955,298.177,-95.304,173.979,32.083,155.873
C09746=1066.949,297.929,-95.274,173.976,32.078,155.873
C09747=1066.943,297.681,-95.242,173.973,32.074,155.872
C09748=1066.937,297.433,-95.210,173.970,32.070,155.871
C09749=1066.931,297.185,-95.179,173.967,32.065,155.870
C09750=1066.925,296.937,-95.147,173.964,32.061,155.869
C09751=1066.919,296.690,-95.116,173.961,32.057,155.869
C09752=1066.912,296.442,-95.084,173.958,32.053,155.868
C09753=1066.907,296.193,-95.053,173.955,32.049,155.867
C09754=1066.901,295.946,-95.022,173.952,32.045,155.866
C09755=1066.895,295.698,-94.990,173.949,32.040,155.865
C09756=1066.888,295.450,-94.959,173.946,32.036,155.865
C09757=1066.882,295.202,-94.928,173.944,32.032,155.864
C09758=1066.876,294.954,-94.896,173.941,32.028,155.863
C09759=1066.870,294.707,-94.865,173.938,32.024,155.862
C09760=1066.864,294.458,-94.834,173.935,32.019,155.862
C09761=1066.858,294.210,-94.802,173.932,32.015,155.861
C09762=1066.851,293.963,-94.771,173.929,32.011,155.860
C09763=1066.845,293.714,-94.741,173.926,32.007,155.859
C09764=1066.840,293.467,-94.709,173.924,32.003,155.859
C09765=1066.833,293.218,-94.678,173.921,31.999,155.858
C09766=1066.827,292.971,-94.647,173.918,31.994,155.857
C09767=1066.821,292.723,-94.615,173.915,31.991,155.856
C09768=1066.815,292.474,-94.584,173.912,31.986,155.855
C09769=1066.809,292.227,-94.553,173.909,31.982,155.855
C09770=1066.802,291.979,-94.523,173.906,31.978,155.854
C09771=1066.797,291.731,-94.491,173.904,31.974,155.853
C09772=1066.790,291.483,-94.460,173.901,31.970,155.852
C09773=1066.784,291.235,-94.429,173.898,31.965,155.852
C09774=1066.779,291.012,-94.402,173.895,31.962,155.851
C09775=1066.774,290.789,-94.374,173.892,31.958,155.850
C09776=1066.768,290.567,-94.346,173.890,31.954,155.850
C09777=1066.762,290.344,-94.318,173.887,31.951,155.849
C09778=1066.757,290.122,-94.290,173.885,31.947,155.848
C09779=1066.752,289.898,-94.263,173.883,31.943,155.848
C09780=1066.746,289.676,-94.235,173.880,31.939,155.847
C09781=1066.740,289.453,-94.207,173.877,31.936,155.846
C09782=1066.735,289.205,-94.176,173.874,31.931,155.845
C09783=1066.728,288.957,-94.145,173.871,31.927,155.845
C09784=1066.723,288.710,-94.115,173.868,31.923,155.844
C09785=1066.716,288.461,-94.084,173.866,31.919,155.843
C09786=1066.710,288.214,-94.053,173.863,31.915,155.842
C09787=1066.704,287.965,-94.022,173.860,31.911,155.842
C09788=1066.698,287.718,-93.992,173.857,31.907,155.841
C09789=1066.691,287.469,-93.961,173.854,31.902,155.840
C09790=1066.685,287.222,-93.930,173.851,31.899,155.839
C09791=1066.679,286.973,-93.899,173.849,31.894,155.839
C09792=1066.673,286.725,-93.869,173.847,31.891,155.838
C09793=1066.667,286.477,-93.838,173.844,31.886,155.837
C09794=1066.661,286.229,-93.808,173.841,31.882,155.836
C09795=1066.655,285.981,-93.778,173.838,31.878,155.836
C09796=1066.649,285.733,-93.747,173.835,31.874,155.835
C09797=1066.642,285.486,-93.716,173.832,31.870,155.834
C09798=1066.636,285.237,-93.685,173.830,31.866,155.833
C09799=1066.630,284.989,-93.655,173.827,31.862,155.833
C09800=1066.624,284.741,-93.624,173.824,31.858,155.832
C09801=1066.618,284.493,-93.594,173.821,31.854,155.831
C09802=1066.612,284.245,-93.563,173.818,31.849,155.830
C09803=1066.606,283.997,-93.533,173.815,31.846,155.830
C09804=1066.600,283.749,-93.502,173.813,31.841,155.829
C09805=1066.594,283.501,-93.472,173.810,31.837,155.828
C09806=1066.588,283.252,-93.441,173.807,31.833,155.827
C09807=1066.581,283.005,-93.411,173.805,31.829,155.827
C09808=1066.575,282.757,-93.381,173.802,31.825,155.826
C09809=1066.569,282.509,-93.351,173.799,31.821,155.825
C09810=1066.563,282.261,-93.320,173.797,31.817,155.824
C09811=1066.557,282.013,-93.290,173.794,31.813,155.824
C09812=1066.552,281.764,-93.260,173.791,31.808,155.823
C09813=1066.545,281.516,-93.229,173.788,31.804,155.822
C09814=1066.540,281.268,-93.199,173.785,31.800,155.821
C09815=1066.534,281.020,-93.169,173.782,31.796,155.821
C09816=1066.528,280.772,-93.138,173.780,31.792,155.820
C09817=1066.521,280.524,-93.108,173.778,31.788,155.819
C09818=1066.515,280.276,-93.078,173.775,31.784,155.818
C09819=1066.509,280.028,-93.048,173.772,31.780,155.818
C09820=1066.503,279.779,-93.017,173.769,31.776,155.817
C09821=1066.497,279.532,-92.987,173.766,31.772,155.816
C09822=1066.491,279.283,-92.958,173.764,31.768,155.815
C09823=1066.485,279.036,-92.928,173.761,31.764,155.815
C09824=1066.479,278.787,-92.897,173.758,31.760,155.814
C09825=1066.472,278.540,-92.867,173.756,31.756,155.813
C09826=1066.467,278.291,-92.838,173.753,31.752,155.812
C09827=1066.461,278.043,-92.807,173.750,31.748,155.812
C09828=1066.454,277.795,-92.777,173.748,31.743,155.811
C09829=1066.448,277.547,-92.748,173.745,31.740,155.810
C09830=1066.444,277.329,-92.721,173.743,31.736,155.810
C09831=1066.438,277.112,-92.695,173.740,31.732,155.809
C09832=1066.432,276.894,-92.669,173.738,31.729,155.808
C09833=1066.427,276.677,-92.642,173.735,31.725,155.808
C09834=1066.422,276.459,-92.616,173.733,31.722,155.807
C09835=1066.416,276.242,-92.590,173.731,31.718,155.806
C09836=1066.411,276.025,-92.563,173.729,31.715,155.806
C09837=1066.405,275.807,-92.537,173.726,31.711,155.805
C09838=1066.400,275.558,-92.507,173.723,31.707,155.804
C09839=1066.393,275.311,-92.478,173.720,31.703,155.804
C09840=1066.388,275.063,-92.448,173.718,31.699,155.803
C09841=1066.382,274.814,-92.419,173.716,31.695,155.802
C09842=1066.376,274.567,-92.389,173.713,31.691,155.802
C09843=1066.370,274.317,-92.359,173.710,31.687,155.801
C09844=1066.363,274.070,-92.329,173.707,31.683,155.800
C09845=1066.358,273.821,-92.299,173.704,31.679,155.799
C09846=1066.351,273.574,-92.269,173.703,31.675,155.799
C09847=1066.346,273.326,-92.240,173.700,31.671,155.798
C09848=1066.340,273.077,-92.210,173.697,31.667,155.797
C09849=1066.334,272.830,-92.180,173.694,31.663,155.796
C09850=1066.327,272.581,-92.151,173.691,31.659,155.796
C09851=1066.321,272.332,-92.121,173.688,31.655,155.795
C09852=1066.315,272.085,-92.092,173.687,31.651,155.794
C09853=1066.309,271.836,-92.062,173.684,31.647,155.793
C09854=1066.303,271.588,-92.033,173.681,31.643,155.793
C09855=1066.297,271.340,-92.003,173.678,31.639,155.792
C09856=1066.291,271.092,-91.974,173.675,31.635,155.791
C09857=1066.285,270.844,-91.944,173.674,31.631,155.791
C09858=1066.279,270.596,-91.915,173.671,31.627,155.790
C09859=1066.273,270.348,-91.886,173.668,31.623,155.789
C09860=1066.267,270.100,-91.856,173.665,31.619,155.788
C09861=1066.261,269.852,-91.826,173.662,31.615,155.788
C09862=1066.255,269.603,-91.797,173.661,31.611,155.787
C09863=1066.248,269.354,-91.767,173.658,31.607,155.786
C09864=1066.242,269.106,-91.738,173.655,31.603,155.786
C09865=1066.237,268.858,-91.709,173.652,31.599,155.785
C09866=1066.230,268.610,-91.679,173.650,31.595,155.784
C09867=1066.224,268.362,-91.650,173.647,31.591,155.783
C09868=1066.218,268.114,-91.620,173.645,31.587,155.783
C09869=1066.212,267.866,-91.591,173.642,31.583,155.782
C09870=1066.206,267.617,-91.562,173.639,31.579,155.781
C09871=1066.200,267.369,-91.533,173.637,31.575,155.781
C09872=1066.194,267.121,-91.504,173.634,31.571,155.780
C09873=1066.188,266.873,-91.475,173.632,31.567,155.779
C09874=1066.182,266.625,-91.446,173.629,31.563,155.778
C09875=1066.176,266.376,-91.416,173.627,31.559,155.778
C09876=1066.170,266.128,-91.387,173.624,31.555,155.777
C09877=1066.164,265.880,-91.358,173.621,31.551,155.776
C09878=1066.157,265.632,-91.329,173.619,31.547,155.776
C09879=1066.152,265.383,-91.299,173.617,31.543,155.775
C09880=1066.145,265.135,-91.270,173.614,31.539,155.774
C09881=1066.140,264.886,-91.242,173.611,31.535,155.773
C09882=1066.133,264.638,-91.213,173.608,31.531,155.773
C09883=1066.128,264.391,-91.183,173.607,31.527,155.772
C09884=1066.122,264.142,-91.154,173.604,31.523,155.771
C09885=1066.116,263.894,-91.125,173.601,31.519,155.771
C09886=1066.111,263.678,-91.100,173.599,31.515,155.770
C09887=1066.105,263.462,-91.076,173.596,31.512,155.769
C09888=1066.099,263.247,-91.050,173.595,31.509,155.769
C09889=1066.095,263.031,-91.024,173.593,31.505,155.768
C09890=1066.089,262.815,-91.000,173.590,31.502,155.767
C09891=1066.084,262.599,-90.975,173.588,31.499,155.767
C09892=1066.079,262.383,-90.950,173.585,31.495,155.766
C09893=1066.073,262.168,-90.924,173.583,31.492,155.766
C09894=1066.067,261.919,-90.896,173.581,31.488,155.765
C09895=1066.060,261.672,-90.867,173.579,31.484,155.764
C09896=1066.054,261.423,-90.838,173.576,31.480,155.763
C09897=1066.048,261.175,-90.810,173.573,31.476,155.763
C09898=1066.042,260.927,-90.781,173.570,31.472,155.762
C09899=1066.035,260.678,-90.752,173.569,31.468,155.761
C09900=1066.029,260.430,-90.724,173.566,31.464,155.761
C09901=1066.024,260.182,-90.695,173.563,31.460,155.760
C09902=1066.018,259.933,-90.667,173.561,31.457,155.759
C09903=1066.012,259.685,-90.638,173.558,31.452,155.759
C09904=1066.005,259.437,-90.609,173.556,31.448,155.758
C09905=1065.999,259.189,-90.581,173.553,31.445,155.757
C09906=1065.992,258.941,-90.552,173.551,31.440,155.756
C09907=1065.987,258.692,-90.523,173.548,31.437,155.756
C09908=1065.980,258.444,-90.494,173.545,31.433,155.755
C09909=1065.975,258.196,-90.466,173.544,31.429,155.754
C09910=1065.969,257.948,-90.437,173.541,31.425,155.754
C09911=1065.963,257.699,-90.409,173.538,31.421,155.753
C09912=1065.956,257.451,-90.380,173.536,31.417,155.752
C09913=1065.950,257.202,-90.352,173.534,31.413,155.752
C09914=1065.944,256.954,-90.323,173.531,31.409,155.751
C09915=1065.938,256.706,-90.295,173.529,31.405,155.750
C09916=1065.932,256.457,-90.267,173.526,31.401,155.749
C09917=1065.926,256.209,-90.238,173.523,31.397,155.749
C09918=1065.920,255.960,-90.210,173.522,31.394,155.748
C09919=1065.913,255.713,-90.181,173.519,31.389,155.747
C09920=1065.908,255.465,-90.153,173.516,31.385,155.747
C09921=1065.902,255.216,-90.125,173.514,31.382,155.746
C09922=1065.896,254.968,-90.096,173.511,31.377,155.745
C09923=1065.890,254.719,-90.068,173.509,31.373,155.745
C09924=1065.884,254.471,-90.040,173.507,31.370,155.744
C09925=1065.877,254.223,-90.011,173.504,31.365,155.743
C09926=1065.871,253.974,-89.983,173.501,31.362,155.742
C09927=1065.865,253.726,-89.954,173.500,31.358,155.742
C09928=1065.860,253.478,-89.927,173.497,31.354,155.741
C09929=1065.854,253.229,-89.897,173.494,31.350,155.740
C09930=1065.847,252.981,-89.870,173.492,31.346,155.739
C09931=1065.842,252.733,-89.842,173.489,31.342,155.739
C09932=1065.836,252.484,-89.813,173.488,31.338,155.738
C09933=1065.830,252.235,-89.785,173.485,31.334,155.737
C09934=1065.824,251.987,-89.756,173.482,31.330,155.737
C09935=1065.818,251.740,-89.729,173.480,31.326,155.736
C09936=1065.812,251.491,-89.700,173.478,31.322,155.735
C09937=1065.806,251.242,-89.672,173.475,31.318,155.735
C09938=1065.800,250.994,-89.644,173.473,31.314,155.734
C09939=1065.794,250.745,-89.616,173.470,31.310,155.733
C09940=1065.788,250.498,-89.588,173.468,31.306,155.732
C09941=1065.782,250.249,-89.559,173.466,31.302,155.732
C09942=1065.776,250.032,-89.535,173.464,31.299,155.731
C09943=1065.772,249.815,-89.510,173.461,31.295,155.730
C09944=1065.767,249.599,-89.486,173.459,31.291,155.730
C09945=1065.761,249.382,-89.461,173.458,31.288,155.729
C09946=1065.756,249.165,-89.437,173.456,31.284,155.729
C09947=1065.751,248.948,-89.413,173.453,31.281,155.728
C09948=1065.746,248.731,-89.388,173.451,31.277,155.727
C09949=1065.741,248.515,-89.364,173.449,31.274,155.727
C09950=1065.735,248.266,-89.335,173.447,31.270,155.726
C09951=1065.729,248.017,-89.308,173.445,31.266,155.725
C09952=1065.723,247.769,-89.280,173.442,31.262,155.725
C09953=1065.717,247.521,-89.251,173.440,31.258,155.724
C09954=1065.712,247.272,-89.223,173.438,31.254,155.723
C09955=1065.705,247.024,-89.196,173.435,31.250,155.722
C09956=1065.700,246.776,-89.168,173.433,31.246,155.722
C09957=1065.694,246.527,-89.139,173.430,31.242,155.721
C09958=1065.688,246.279,-89.113,173.428,31.238,155.720
C09959=1065.682,246.030,-89.084,173.426,31.234,155.720
C09960=1065.676,245.782,-89.057,173.423,31.230,155.719
C09961=1065.670,245.534,-89.029,173.421,31.226,155.718
C09962=1065.664,245.285,-89.001,173.418,31.222,155.717
C09963=1065.658,245.037,-88.973,173.417,31.218,155.717
C09964=1065.652,244.788,-88.946,173.414,31.214,155.716
C09965=1065.647,244.540,-88.918,173.412,31.210,155.715
C09966=1065.640,244.292,-88.890,173.409,31.206,155.715
C09967=1065.635,244.044,-88.862,173.408,31.202,155.714
C09968=1065.628,243.794,-88.835,173.405,31.198,155.713
C09969=1065.623,243.546,-88.807,173.402,31.194,155.712
C09970=1065.616,243.298,-88.780,173.400,31.190,155.712
C09971=1065.611,243.050,-88.752,173.398,31.186,155.711
C09972=1065.604,242.801,-88.725,173.396,31.182,155.710
C09973=1065.599,242.553,-88.697,173.393,31.178,155.710
C09974=1065.592,242.304,-88.669,173.391,31.174,155.709
C09975=1065.587,242.056,-88.642,173.389,31.170,155.708
C09976=1065.581,241.807,-88.614,173.387,31.166,155.708
C09977=1065.574,241.558,-88.587,173.384,31.162,155.707
C09978=1065.568,241.310,-88.560,173.382,31.158,155.706
C09979=1065.562,241.062,-88.532,173.380,31.154,155.705
C09980=1065.556,240.813,-88.505,173.377,31.150,155.705
C09981=1065.550,240.565,-88.477,173.375,31.146,155.704
C09982=1065.544,240.317,-88.450,173.372,31.142,155.703
C09983=1065.538,240.068,-88.422,173.371,31.138,155.703
C09984=1065.532,239.819,-88.395,173.368,31.134,155.702
C09985=1065.526,239.572,-88.368,173.366,31.131,155.701
C09986=1065.520,239.323,-88.341,173.363,31.126,155.700
C09987=1065.515,239.075,-88.313,173.362,31.122,155.700
C09988=1065.508,238.826,-88.286,173.359,31.119,155.699
C09989=1065.502,238.578,-88.259,173.357,31.114,155.698
C09990=1065.496,238.329,-88.232,173.354,31.110,155.698
C09991=1065.490,238.081,-88.204,173.353,31.107,155.697
C09992=1065.483,237.832,-88.177,173.350,31.102,155.696
C09993=1065.478,237.583,-88.150,173.348,31.099,155.696
C09994=1065.472,237.335,-88.123,173.345,31.095,155.695
C09995=1065.466,237.086,-88.096,173.344,31.091,155.694
C09996=1065.460,236.839,-88.068,173.341,31.087,155.693
//INST
///DATE 2021/06/17 10:55
///ATTR SC,RW,RJ
////FRAME ROBOT
///GROUP1 RB1
NOP
MOVL C00000 V=800.0 PL=0
MOVL C00001 V=800.0 PL=0
MOVL C00002 V=800.0 PL=0
MOVL C00003 V=800.0 PL=0
MOVL C00004 V=800.0 PL=0
MOVL C00005 V=800.0 PL=0
MOVL C00006 V=800.0 PL=0
MOVL C00007 V=800.0 PL=0
MOVL C00008 V=800.0 PL=0
MOVL C00009 V=800.0 PL=0
MOVL C00010 V=800.0 PL=0
MOVL C00011 V=800.0 PL=0
MOVL C00012 V=800.0 PL=0
MOVL C00013 V=800.0 PL=0
MOVL C00014 V=800.0 PL=0
MOVL C00015 V=800.0 PL=0
MOVL C00016 V=800.0 PL=0
MOVL C00017 V=800.0 PL=0
MOVL C00018 V=800.0 PL=0
MOVL C00019 V=800.0 PL=0
MOVL C00020 V=800.0 PL=0
MOVL C00021 V=800.0 PL=0
MOVL C00022 V=800.0 PL=0
MOVL C00023 V=800.0 PL=0
MOVL C00024 V=800.0 PL=0
MOVL C00025 V=800.0 PL=0
MOVL C00026 V=800.0 PL=0
MOVL C00027 V=800.0 PL=0
MOVL C00028 V=800.0 PL=0
MOVL C00029 V=800.0 PL=0
MOVL C00030 V=800.0 PL=0
MOVL C00031 V=800.0 PL=0
MOVL C00032 V=800.0 PL=0
MOVL C00033 V=800.0 PL=0
MOVL C00034 V=800.0 PL=0
MOVL C00035 V=800.0 PL=0
MOVL C00036 V=800.0 PL=0
MOVL C00037 V=800.0 PL=0
MOVL C00038 V=800.0 PL=0
MOVL C00039 V=800.0 PL=0
MOVL C00040 V=800.0 PL=0
MOVL C00041 V=800.0 PL=0
MOVL C00042 V=800.0 PL=0
MOVL C00043 V=800.0 PL=0
MOVL C00044 V=800.0 PL=0
MOVL C00045 V=800.0 PL=0
MOVL C00046 V=800.0 PL=0
MOVL C00047 V=800.0 PL=0
MOVL C00048 V=800.0 PL=0
MOVL C00049 V=800.0 PL=0
MOVL C00050 V=800.0 PL=0
MOVL C00051 V=800.0 PL=0
MOVL C00052 V=800.0 PL=0
MOVL C00053 V=800.0 PL=0
MOVL C00054 V=800.0 PL=0
MOVL C00055 V=800.0 PL=0
MOVL C00056 V=800.0 PL=0
MOVL C00057 V=800.0 PL=0
MOVL C00058 V=800.0 PL=0
MOVL C00059 V=800.0 PL=0
MOVL C00060 V=800.0 PL=0
MOVL C00061 V=800.0 PL=0
MOVL C00062 V=800.0 PL=0
MOVL C00063 V=800.0 PL=0
MOVL C00064 V=800.0 PL=0
MOVL C00065 V=800.0 PL=0
MOVL C00066 V=800.0 PL=0
MOVL C00067 V=800.0 PL=0
MOVL C00068 V=800.0 PL=0
MOVL C00069 V=800.0 PL=0
MOVL C00070 V=800.0 PL=0
MOVL C00071 V=800.0 PL=0
MOVL C00072 V=800.0 PL=0
MOVL C00073 V=800.0 PL=0
MOVL C00074 V=800.0 PL=0
MOVL C00075 V=800.0 PL=0
MOVL C00076 V=800.0 PL=0
MOVL C00077 V=800.0 PL=0
MOVL C00078 V=800.0 PL=0
MOVL C00079 V=800.0 PL=0
MOVL C00080 V=800.0 PL=0
MOVL C00081 V=800.0 PL=0
MOVL C00082 V=800.0 PL=0
MOVL C00083 V=800.0 PL=0
MOVL C00084 V=800.0 PL=0
MOVL C00085 V=800.0 PL=0
MOVL C00086 V=800.0 PL=0
MOVL C00087 V=800.0 PL=0
MOVL C00088 V=800.0 PL=0
MOVL C00089 V=800.0 PL=0
MOVL C00090 V=800.0 PL=0
MOVL C00091 V=800.0 PL=0
MOVL C00092 V=800.0 PL=0
MOVL C00093 V=800.0 PL=0
MOVL C00094 V=800.0 PL=0
MOVL C00095 V=800.0 PL=0
MOVL C00096 V=800.0 PL=0
MOVL C00097 V=800.0 PL=0
MOVL C00098 V=800.0 PL=0
MOVL C00099 V=800.0 PL=0
MOVL C00100 V=800.0 PL=0
MOVL C00101 V=800.0 PL=0
MOVL C00102 V=800.0 PL=0
MOVL C00103 V=800.0 PL=0
MOVL C00104 V=800.0 PL=0
MOVL C00105 V=800.0 PL=0
MOVL C00106 V=800.0 PL=0
MOVL C00107 V=800.0 PL=0
MOVL C00108 V=800.0 PL=0
MOVL C00109 V=800.0 PL=0
MOVL C00110 V=800.0 PL=0
MOVL C00111 V=800.0 PL=0
MOVL C00112 V=800.0 PL=0
MOVL C00113 V=800.0 PL=0
MOVL C00114 V=800.0 PL=0
MOVL C00115 V=800.0 PL=0
MOVL C00116 V=800.0 PL=0
MOVL C00117 V=800.0 PL=0
MOVL C00118 V=800.0 PL=0
MOVL C00119 V=800.0 PL=0
MOVL C00120 V=800.0 PL=0
MOVL C00121 V=800.0 PL=0
MOVL C00122 V=800.0 PL=0
MOVL C00123 V=800.0 PL=0
MOVL C00124 V=800.0 PL=0
MOVL C00125 V=800.0 PL=0
MOVL C00126 V=800.0 PL=0
MOVL C00127 V=800.0 PL=0
MOVL C00128 V=800.0 PL=0
MOVL C00129 V=800.0 PL=0
MOVL C00130 V=800.0 PL=0
MOVL C00131 V=800.0 PL=0
MOVL C00132 V=800.0 PL=0
MOVL C00133 V=800.0 PL=0
MOVL C00134 V=800.0 PL=0
MOVL C00135 V=800.0 PL=0
MOVL C00136 V=800.0 PL=0
MOVL C00137 V=800.0 PL=0
MOVL C00138 V=800.0 PL=0
MOVL C00139 V=800.0 PL=0
MOVL C00140 V=800.0 PL=0
MOVL C00141 V=800.0 PL=0
MOVL C00142 V=800.0 PL=0
MOVL C00143 V=800.0 PL=0
MOVL C00144 V=800.0 PL=0
MOVL C00145 V=800.0 PL=0
MOVL C00146 V=800.0 PL=0
MOVL C00147 V=800.0 PL=0
MOVL C00148 V=800.0 PL=0
MOVL C00149 V=800.0 PL=0
MOVL C00150 V=800.0 PL=0
MOVL C00151 V=800.0 PL=0
MOVL C00152 V=800.0 PL=0
MOVL C00153 V=800.0 PL=0
MOVL C00154 V=800.0 PL=0
MOVL C00155 V=800.0 PL=0
MOVL C00156 V=800.0 PL=0
MOVL C00157 V=800.0 PL=0
MOVL C00158 V=800.0 PL=0
MOVL C00159 V=800.0 PL=0
MOVL C00160 V=800.0 PL=0
MOVL C00161 V=800.0 PL=0
MOVL C00162 V=800.0 PL=0
MOVL C00163 V=800.0 PL=0
MOVL C00164 V=800.0 PL=0
MOVL C00165 V=800.0 PL=0
MOVL C00166 V=800.0 PL=0
MOVL C00167 V=800.0 PL=0
MOVL C00168 V=800.0 PL=0
MOVL C00169 V=800.0 PL=0
MOVL C00170 V=800.0 PL=0
MOVL C00171 V=800.0 PL=0
MOVL C00172 V=800.0 PL=0
MOVL C00173 V=800.0 PL=0
MOVL C00174 V=800.0 PL=0
MOVL C00175 V=800.0 PL=0
MOVL C00176 V=800.0 PL=0
MOVL C00177 V=800.0 PL=0
MOVL C00178 V=800.0 PL=0
MOVL C00179 V=800.0 PL=0
MOVL C00180 V=800.0 PL=0
MOVL C00181 V=800.0 PL=0
MOVL C00182 V=800.0 PL=0
MOVL C00183 V=800.0 PL=0
MOVL C00184 V=800.0 PL=0
MOVL C00185 V=800.0 PL=0
MOVL C00186 V=800.0 PL=0
MOVL C00187 V=800.0 PL=0
MOVL C00188 V=800.0 PL=0
MOVL C00189 V=800.0 PL=0
MOVL C00190 V=800.0 PL=0
MOVL C00191 V=800.0 PL=0
MOVL C00192 V=800.0 PL=0
MOVL C00193 V=800.0 PL=0
MOVL C00194 V=800.0 PL=0
MOVL C00195 V=800.0 PL=0
MOVL C00196 V=800.0 PL=0
MOVL C00197 V=800.0 PL=0
MOVL C00198 V=800.0 PL=0
MOVL C00199 V=800.0 PL=0
MOVL C00200 V=800.0 PL=0
MOVL C00201 V=800.0 PL=0
MOVL C00202 V=800.0 PL=0
MOVL C00203 V=800.0 PL=0
MOVL C00204 V=800.0 PL=0
MOVL C00205 V=800.0 PL=0
MOVL C00206 V=800.0 PL=0
MOVL C00207 V=800.0 PL=0
MOVL C00208 V=800.0 PL=0
MOVL C00209 V=800.0 PL=0
MOVL C00210 V=800.0 PL=0
MOVL C00211 V=800.0 PL=0
MOVL C00212 V=800.0 PL=0
MOVL C00213 V=800.0 PL=0
MOVL C00214 V=800.0 PL=0
MOVL C00215 V=800.0 PL=0
MOVL C00216 V=800.0 PL=0
MOVL C00217 V=800.0 PL=0
MOVL C00218 V=800.0 PL=0
MOVL C00219 V=800.0 PL=0
MOVL C00220 V=800.0 PL=0
MOVL C00221 V=800.0 PL=0
MOVL C00222 V=800.0 PL=0
MOVL C00223 V=800.0 PL=0
MOVL C00224 V=800.0 PL=0
MOVL C00225 V=800.0 PL=0
MOVL C00226 V=800.0 PL=0
MOVL C00227 V=800.0 PL=0
MOVL C00228 V=800.0 PL=0
MOVL C00229 V=800.0 PL=0
MOVL C00230 V=800.0 PL=0
MOVL C00231 V=800.0 PL=0
MOVL C00232 V=800.0 PL=0
MOVL C00233 V=800.0 PL=0
MOVL C00234 V=800.0 PL=0
MOVL C00235 V=800.0 PL=0
MOVL C00236 V=800.0 PL=0
MOVL C00237 V=800.0 PL=0
MOVL C00238 V=800.0 PL=0
MOVL C00239 V=800.0 PL=0
MOVL C00240 V=800.0 PL=0
MOVL C00241 V=800.0 PL=0
MOVL C00242 V=800.0 PL=0
MOVL C00243 V=800.0 PL=0
MOVL C00244 V=800.0 PL=0
MOVL C00245 V=800.0 PL=0
MOVL C00246 V=800.0 PL=0
MOVL C00247 V=800.0 PL=0
MOVL C00248 V=800.0 PL=0
MOVL C00249 V=800.0 PL=0
MOVL C00250 V=800.0 PL=0
MOVL C00251 V=800.0 PL=0
MOVL C00252 V=800.0 PL=0
MOVL C00253 V=800.0 PL=0
MOVL C00254 V=800.0 PL=0
MOVL C00255 V=800.0 PL=0
MOVL C00256 V=800.0 PL=0
MOVL C00257 V=800.0 PL=0
MOVL C00258 V=800.0 PL=0
MOVL C00259 V=800.0 PL=0
MOVL C00260 V=800.0 PL=0
MOVL C00261 V=800.0 PL=0
MOVL C00262 V=800.0 PL=0
MOVL C00263 V=800.0 PL=0
MOVL C00264 V=800.0 PL=0
MOVL C00265 V=800.0 PL=0
MOVL C00266 V=800.0 PL=0
MOVL C00267 V=800.0 PL=0
MOVL C00268 V=800.0 PL=0
MOVL C00269 V=800.0 PL=0
MOVL C00270 V=800.0 PL=0
MOVL C00271 V=800.0 PL=0
MOVL C00272 V=800.0 PL=0
MOVL C00273 V=800.0 PL=0
MOVL C00274 V=800.0 PL=0
MOVL C00275 V=800.0 PL=0
MOVL C00276 V=800.0 PL=0
MOVL C00277 V=800.0 PL=0
MOVL C00278 V=800.0 PL=0
MOVL C00279 V=800.0 PL=0
MOVL C00280 V=800.0 PL=0
MOVL C00281 V=800.0 PL=0
MOVL C00282 V=800.0 PL=0
MOVL C00283 V=800.0 PL=0
MOVL C00284 V=800.0 PL=0
MOVL C00285 V=800.0 PL=0
MOVL C00286 V=800.0 PL=0
MOVL C00287 V=800.0 PL=0
MOVL C00288 V=800.0 PL=0
MOVL C00289 V=800.0 PL=0
MOVL C00290 V=800.0 PL=0
MOVL C00291 V=800.0 PL=0
MOVL C00292 V=800.0 PL=0
MOVL C00293 V=800.0 PL=0
MOVL C00294 V=800.0 PL=0
MOVL C00295 V=800.0 PL=0
MOVL C00296 V=800.0 PL=0
MOVL C00297 V=800.0 PL=0
MOVL C00298 V=800.0 PL=0
MOVL C00299 V=800.0 PL=0
MOVL C00300 V=800.0 PL=0
MOVL C00301 V=800.0 PL=0
MOVL C00302 V=800.0 PL=0
MOVL C00303 V=800.0 PL=0
MOVL C00304 V=800.0 PL=0
MOVL C00305 V=800.0 PL=0
MOVL C00306 V=800.0 PL=0
MOVL C00307 V=800.0 PL=0
MOVL C00308 V=800.0 PL=0
MOVL C00309 V=800.0 PL=0
MOVL C00310 V=800.0 PL=0
MOVL C00311 V=800.0 PL=0
MOVL C00312 V=800.0 PL=0
MOVL C00313 V=800.0 PL=0
MOVL C00314 V=800.0 PL=0
MOVL C00315 V=800.0 PL=0
MOVL C00316 V=800.0 PL=0
MOVL C00317 V=800.0 PL=0
MOVL C00318 V=800.0 PL=0
MOVL C00319 V=800.0 PL=0
MOVL C00320 V=800.0 PL=0
MOVL C00321 V=800.0 PL=0
MOVL C00322 V=800.0 PL=0
MOVL C00323 V=800.0 PL=0
MOVL C00324 V=800.0 PL=0
MOVL C00325 V=800.0 PL=0
MOVL C00326 V=800.0 PL=0
MOVL C00327 V=800.0 PL=0
MOVL C00328 V=800.0 PL=0
MOVL C00329 V=800.0 PL=0
MOVL C00330 V=800.0 PL=0
MOVL C00331 V=800.0 PL=0
MOVL C00332 V=800.0 PL=0
MOVL C00333 V=800.0 PL=0
MOVL C00334 V=800.0 PL=0
MOVL C00335 V=800.0 PL=0
MOVL C00336 V=800.0 PL=0
MOVL C00337 V=800.0 PL=0
MOVL C00338 V=800.0 PL=0
MOVL C00339 V=800.0 PL=0
MOVL C00340 V=800.0 PL=0
MOVL C00341 V=800.0 PL=0
MOVL C00342 V=800.0 PL=0
MOVL C00343 V=800.0 PL=0
MOVL C00344 V=800.0 PL=0
MOVL C00345 V=800.0 PL=0
MOVL C00346 V=800.0 PL=0
MOVL C00347 V=800.0 PL=0
MOVL C00348 V=800.0 PL=0
MOVL C00349 V=800.0 PL=0
MOVL C00350 V=800.0 PL=0
MOVL C00351 V=800.0 PL=0
MOVL C00352 V=800.0 PL=0
MOVL C00353 V=800.0 PL=0
MOVL C00354 V=800.0 PL=0
MOVL C00355 V=800.0 PL=0
MOVL C00356 V=800.0 PL=0
MOVL C00357 V=800.0 PL=0
MOVL C00358 V=800.0 PL=0
MOVL C00359 V=800.0 PL=0
MOVL C00360 V=800.0 PL=0
MOVL C00361 V=800.0 PL=0
MOVL C00362 V=800.0 PL=0
MOVL C00363 V=800.0 PL=0
MOVL C00364 V=800.0 PL=0
MOVL C00365 V=800.0 PL=0
MOVL C00366 V=800.0 PL=0
MOVL C00367 V=800.0 PL=0
MOVL C00368 V=800.0 PL=0
MOVL C00369 V=800.0 PL=0
MOVL C00370 V=800.0 PL=0
MOVL C00371 V=800.0 PL=0
MOVL C00372 V=800.0 PL=0
MOVL C00373 V=800.0 PL=0
MOVL C00374 V=800.0 PL=0
MOVL C00375 V=800.0 PL=0
MOVL C00376 V=800.0 PL=0
MOVL C00377 V=800.0 PL=0
MOVL C00378 V=800.0 PL=0
MOVL C00379 V=800.0 PL=0
MOVL C00380 V=800.0 PL=0
MOVL C00381 V=800.0 PL=0
MOVL C00382 V=800.0 PL=0
MOVL C00383 V=800.0 PL=0
MOVL C00384 V=800.0 PL=0
MOVL C00385 V=800.0 PL=0
MOVL C00386 V=800.0 PL=0
MOVL C00387 V=800.0 PL=0
MOVL C00388 V=800.0 PL=0
MOVL C00389 V=800.0 PL=0
MOVL C00390 V=800.0 PL=0
MOVL C00391 V=800.0 PL=0
MOVL C00392 V=800.0 PL=0
MOVL C00393 V=800.0 PL=0
MOVL C00394 V=800.0 PL=0
MOVL C00395 V=800.0 PL=0
MOVL C00396 V=800.0 PL=0
MOVL C00397 V=800.0 PL=0
MOVL C00398 V=800.0 PL=0
MOVL C00399 V=800.0 PL=0
MOVL C00400 V=800.0 PL=0
MOVL C00401 V=800.0 PL=0
MOVL C00402 V=800.0 PL=0
MOVL C00403 V=800.0 PL=0
MOVL C00404 V=800.0 PL=0
MOVL C00405 V=800.0 PL=0
MOVL C00406 V=800.0 PL=0
MOVL C00407 V=800.0 PL=0
MOVL C00408 V=800.0 PL=0
MOVL C00409 V=800.0 PL=0
MOVL C00410 V=800.0 PL=0
MOVL C00411 V=800.0 PL=0
MOVL C00412 V=800.0 PL=0
MOVL C00413 V=800.0 PL=0
MOVL C00414 V=800.0 PL=0
MOVL C00415 V=800.0 PL=0
MOVL C00416 V=800.0 PL=0
MOVL C00417 V=800.0 PL=0
MOVL C00418 V=800.0 PL=0
MOVL C00419 V=800.0 PL=0
MOVL C00420 V=800.0 PL=0
MOVL C00421 V=800.0 PL=0
MOVL C00422 V=800.0 PL=0
MOVL C00423 V=800.0 PL=0
MOVL C00424 V=800.0 PL=0
MOVL C00425 V=800.0 PL=0
MOVL C00426 V=800.0 PL=0
MOVL C00427 V=800.0 PL=0
MOVL C00428 V=800.0 PL=0
MOVL C00429 V=800.0 PL=0
MOVL C00430 V=800.0 PL=0
MOVL C00431 V=800.0 PL=0
MOVL C00432 V=800.0 PL=0
MOVL C00433 V=800.0 PL=0
MOVL C00434 V=800.0 PL=0
MOVL C00435 V=800.0 PL=0
MOVL C00436 V=800.0 PL=0
MOVL C00437 V=800.0 PL=0
MOVL C00438 V=800.0 PL=0
MOVL C00439 V=800.0 PL=0
MOVL C00440 V=800.0 PL=0
MOVL C00441 V=800.0 PL=0
MOVL C00442 V=800.0 PL=0
MOVL C00443 V=800.0 PL=0
MOVL C00444 V=800.0 PL=0
MOVL C00445 V=800.0 PL=0
MOVL C00446 V=800.0 PL=0
MOVL C00447 V=800.0 PL=0
MOVL C00448 V=800.0 PL=0
MOVL C00449 V=800.0 PL=0
MOVL C00450 V=800.0 PL=0
MOVL C00451 V=800.0 PL=0
MOVL C00452 V=800.0 PL=0
MOVL C00453 V=800.0 PL=0
MOVL C00454 V=800.0 PL=0
MOVL C00455 V=800.0 PL=0
MOVL C00456 V=800.0 PL=0
MOVL C00457 V=800.0 PL=0
MOVL C00458 V=800.0 PL=0
MOVL C00459 V=800.0 PL=0
MOVL C00460 V=800.0 PL=0
MOVL C00461 V=800.0 PL=0
MOVL C00462 V=800.0 PL=0
MOVL C00463 V=800.0 PL=0
MOVL C00464 V=800.0 PL=0
MOVL C00465 V=800.0 PL=0
MOVL C00466 V=800.0 PL=0
MOVL C00467 V=800.0 PL=0
MOVL C00468 V=800.0 PL=0
MOVL C00469 V=800.0 PL=0
MOVL C00470 V=800.0 PL=0
MOVL C00471 V=800.0 PL=0
MOVL C00472 V=800.0 PL=0
MOVL C00473 V=800.0 PL=0
MOVL C00474 V=800.0 PL=0
MOVL C00475 V=800.0 PL=0
MOVL C00476 V=800.0 PL=0
MOVL C00477 V=800.0 PL=0
MOVL C00478 V=800.0 PL=0
MOVL C00479 V=800.0 PL=0
MOVL C00480 V=800.0 PL=0
MOVL C00481 V=800.0 PL=0
MOVL C00482 V=800.0 PL=0
MOVL C00483 V=800.0 PL=0
MOVL C00484 V=800.0 PL=0
MOVL C00485 V=800.0 PL=0
MOVL C00486 V=800.0 PL=0
MOVL C00487 V=800.0 PL=0
MOVL C00488 V=800.0 PL=0
MOVL C00489 V=800.0 PL=0
MOVL C00490 V=800.0 PL=0
MOVL C00491 V=800.0 PL=0
MOVL C00492 V=800.0 PL=0
MOVL C00493 V=800.0 PL=0
MOVL C00494 V=800.0 PL=0
MOVL C00495 V=800.0 PL=0
MOVL C00496 V=800.0 PL=0
MOVL C00497 V=800.0 PL=0
MOVL C00498 V=800.0 PL=0
MOVL C00499 V=800.0 PL=0
MOVL C00500 V=800.0 PL=0
MOVL C00501 V=800.0 PL=0
MOVL C00502 V=800.0 PL=0
MOVL C00503 V=800.0 PL=0
MOVL C00504 V=800.0 PL=0
MOVL C00505 V=800.0 PL=0
MOVL C00506 V=800.0 PL=0
MOVL C00507 V=800.0 PL=0
MOVL C00508 V=800.0 PL=0
MOVL C00509 V=800.0 PL=0
MOVL C00510 V=800.0 PL=0
MOVL C00511 V=800.0 PL=0
MOVL C00512 V=800.0 PL=0
MOVL C00513 V=800.0 PL=0
MOVL C00514 V=800.0 PL=0
MOVL C00515 V=800.0 PL=0
MOVL C00516 V=800.0 PL=0
MOVL C00517 V=800.0 PL=0
MOVL C00518 V=800.0 PL=0
MOVL C00519 V=800.0 PL=0
MOVL C00520 V=800.0 PL=0
MOVL C00521 V=800.0 PL=0
MOVL C00522 V=800.0 PL=0
MOVL C00523 V=800.0 PL=0
MOVL C00524 V=800.0 PL=0
MOVL C00525 V=800.0 PL=0
MOVL C00526 V=800.0 PL=0
MOVL C00527 V=800.0 PL=0
MOVL C00528 V=800.0 PL=0
MOVL C00529 V=800.0 PL=0
MOVL C00530 V=800.0 PL=0
MOVL C00531 V=800.0 PL=0
MOVL C00532 V=800.0 PL=0
MOVL C00533 V=800.0 PL=0
MOVL C00534 V=800.0 PL=0
MOVL C00535 V=800.0 PL=0
MOVL C00536 V=800.0 PL=0
MOVL C00537 V=800.0 PL=0
MOVL C00538 V=800.0 PL=0
MOVL C00539 V=800.0 PL=0
MOVL C00540 V=800.0 PL=0
MOVL C00541 V=800.0 PL=0
MOVL C00542 V=800.0 PL=0
MOVL C00543 V=800.0 PL=0
MOVL C00544 V=800.0 PL=0
MOVL C00545 V=800.0 PL=0
MOVL C00546 V=800.0 PL=0
MOVL C00547 V=800.0 PL=0
MOVL C00548 V=800.0 PL=0
MOVL C00549 V=800.0 PL=0
MOVL C00550 V=800.0 PL=0
MOVL C00551 V=800.0 PL=0
MOVL C00552 V=800.0 PL=0
MOVL C00553 V=800.0 PL=0
MOVL C00554 V=800.0 PL=0
MOVL C00555 V=800.0 PL=0
MOVL C00556 V=800.0 PL=0
MOVL C00557 V=800.0 PL=0
MOVL C00558 V=800.0 PL=0
MOVL C00559 V=800.0 PL=0
MOVL C00560 V=800.0 PL=0
MOVL C00561 V=800.0 PL=0
MOVL C00562 V=800.0 PL=0
MOVL C00563 V=800.0 PL=0
MOVL C00564 V=800.0 PL=0
MOVL C00565 V=800.0 PL=0
MOVL C00566 V=800.0 PL=0
MOVL C00567 V=800.0 PL=0
MOVL C00568 V=800.0 PL=0
MOVL C00569 V=800.0 PL=0
MOVL C00570 V=800.0 PL=0
MOVL C00571 V=800.0 PL=0
MOVL C00572 V=800.0 PL=0
MOVL C00573 V=800.0 PL=0
MOVL C00574 V=800.0 PL=0
MOVL C00575 V=800.0 PL=0
MOVL C00576 V=800.0 PL=0
MOVL C00577 V=800.0 PL=0
MOVL C00578 V=800.0 PL=0
MOVL C00579 V=800.0 PL=0
MOVL C00580 V=800.0 PL=0
MOVL C00581 V=800.0 PL=0
MOVL C00582 V=800.0 PL=0
MOVL C00583 V=800.0 PL=0
MOVL C00584 V=800.0 PL=0
MOVL C00585 V=800.0 PL=0
MOVL C00586 V=800.0 PL=0
MOVL C00587 V=800.0 PL=0
MOVL C00588 V=800.0 PL=0
MOVL C00589 V=800.0 PL=0
MOVL C00590 V=800.0 PL=0
MOVL C00591 V=800.0 PL=0
MOVL C00592 V=800.0 PL=0
MOVL C00593 V=800.0 PL=0
MOVL C00594 V=800.0 PL=0
MOVL C00595 V=800.0 PL=0
MOVL C00596 V=800.0 PL=0
MOVL C00597 V=800.0 PL=0
MOVL C00598 V=800.0 PL=0
MOVL C00599 V=800.0 PL=0
MOVL C00600 V=800.0 PL=0
MOVL C00601 V=800.0 PL=0
MOVL C00602 V=800.0 PL=0
MOVL C00603 V=800.0 PL=0
MOVL C00604 V=800.0 PL=0
MOVL C00605 V=800.0 PL=0
MOVL C00606 V=800.0 PL=0
MOVL C00607 V=800.0 PL=0
MOVL C00608 V=800.0 PL=0
MOVL C00609 V=800.0 PL=0
MOVL C00610 V=800.0 PL=0
MOVL C00611 V=800.0 PL=0
MOVL C00612 V=800.0 PL=0
MOVL C00613 V=800.0 PL=0
MOVL C00614 V=800.0 PL=0
MOVL C00615 V=800.0 PL=0
MOVL C00616 V=800.0 PL=0
MOVL C00617 V=800.0 PL=0
MOVL C00618 V=800.0 PL=0
MOVL C00619 V=800.0 PL=0
MOVL C00620 V=800.0 PL=0
MOVL C00621 V=800.0 PL=0
MOVL C00622 V=800.0 PL=0
MOVL C00623 V=800.0 PL=0
MOVL C00624 V=800.0 PL=0
MOVL C00625 V=800.0 PL=0
MOVL C00626 V=800.0 PL=0
MOVL C00627 V=800.0 PL=0
MOVL C00628 V=800.0 PL=0
MOVL C00629 V=800.0 PL=0
MOVL C00630 V=800.0 PL=0
MOVL C00631 V=800.0 PL=0
MOVL C00632 V=800.0 PL=0
MOVL C00633 V=800.0 PL=0
MOVL C00634 V=800.0 PL=0
MOVL C00635 V=800.0 PL=0
MOVL C00636 V=800.0 PL=0
MOVL C00637 V=800.0 PL=0
MOVL C00638 V=800.0 PL=0
MOVL C00639 V=800.0 PL=0
MOVL C00640 V=800.0 PL=0
MOVL C00641 V=800.0 PL=0
MOVL C00642 V=800.0 PL=0
MOVL C00643 V=800.0 PL=0
MOVL C00644 V=800.0 PL=0
MOVL C00645 V=800.0 PL=0
MOVL C00646 V=800.0 PL=0
MOVL C00647 V=800.0 PL=0
MOVL C00648 V=800.0 PL=0
MOVL C00649 V=800.0 PL=0
MOVL C00650 V=800.0 PL=0
MOVL C00651 V=800.0 PL=0
MOVL C00652 V=800.0 PL=0
MOVL C00653 V=800.0 PL=0
MOVL C00654 V=800.0 PL=0
MOVL C00655 V=800.0 PL=0
MOVL C00656 V=800.0 PL=0
MOVL C00657 V=800.0 PL=0
MOVL C00658 V=800.0 PL=0
MOVL C00659 V=800.0 PL=0
MOVL C00660 V=800.0 PL=0
MOVL C00661 V=800.0 PL=0
MOVL C00662 V=800.0 PL=0
MOVL C00663 V=800.0 PL=0
MOVL C00664 V=800.0 PL=0
MOVL C00665 V=800.0 PL=0
MOVL C00666 V=800.0 PL=0
MOVL C00667 V=800.0 PL=0
MOVL C00668 V=800.0 PL=0
MOVL C00669 V=800.0 PL=0
MOVL C00670 V=800.0 PL=0
MOVL C00671 V=800.0 PL=0
MOVL C00672 V=800.0 PL=0
MOVL C00673 V=800.0 PL=0
MOVL C00674 V=800.0 PL=0
MOVL C00675 V=800.0 PL=0
MOVL C00676 V=800.0 PL=0
MOVL C00677 V=800.0 PL=0
MOVL C00678 V=800.0 PL=0
MOVL C00679 V=800.0 PL=0
MOVL C00680 V=800.0 PL=0
MOVL C00681 V=800.0 PL=0
MOVL C00682 V=800.0 PL=0
MOVL C00683 V=800.0 PL=0
MOVL C00684 V=800.0 PL=0
MOVL C00685 V=800.0 PL=0
MOVL C00686 V=800.0 PL=0
MOVL C00687 V=800.0 PL=0
MOVL C00688 V=800.0 PL=0
MOVL C00689 V=800.0 PL=0
MOVL C00690 V=800.0 PL=0
MOVL C00691 V=800.0 PL=0
MOVL C00692 V=800.0 PL=0
MOVL C00693 V=800.0 PL=0
MOVL C00694 V=800.0 PL=0
MOVL C00695 V=800.0 PL=0
MOVL C00696 V=800.0 PL=0
MOVL C00697 V=800.0 PL=0
MOVL C00698 V=800.0 PL=0
MOVL C00699 V=800.0 PL=0
MOVL C00700 V=800.0 PL=0
MOVL C00701 V=800.0 PL=0
MOVL C00702 V=800.0 PL=0
MOVL C00703 V=800.0 PL=0
MOVL C00704 V=800.0 PL=0
MOVL C00705 V=800.0 PL=0
MOVL C00706 V=800.0 PL=0
MOVL C00707 V=800.0 PL=0
MOVL C00708 V=800.0 PL=0
MOVL C00709 V=800.0 PL=0
MOVL C00710 V=800.0 PL=0
MOVL C00711 V=800.0 PL=0
MOVL C00712 V=800.0 PL=0
MOVL C00713 V=800.0 PL=0
MOVL C00714 V=800.0 PL=0
MOVL C00715 V=800.0 PL=0
MOVL C00716 V=800.0 PL=0
MOVL C00717 V=800.0 PL=0
MOVL C00718 V=800.0 PL=0
MOVL C00719 V=800.0 PL=0
MOVL C00720 V=800.0 PL=0
MOVL C00721 V=800.0 PL=0
MOVL C00722 V=800.0 PL=0
MOVL C00723 V=800.0 PL=0
MOVL C00724 V=800.0 PL=0
MOVL C00725 V=800.0 PL=0
MOVL C00726 V=800.0 PL=0
MOVL C00727 V=800.0 PL=0
MOVL C00728 V=800.0 PL=0
MOVL C00729 V=800.0 PL=0
MOVL C00730 V=800.0 PL=0
MOVL C00731 V=800.0 PL=0
MOVL C00732 V=800.0 PL=0
MOVL C00733 V=800.0 PL=0
MOVL C00734 V=800.0 PL=0
MOVL C00735 V=800.0 PL=0
MOVL C00736 V=800.0 PL=0
MOVL C00737 V=800.0 PL=0
MOVL C00738 V=800.0 PL=0
MOVL C00739 V=800.0 PL=0
MOVL C00740 V=800.0 PL=0
MOVL C00741 V=800.0 PL=0
MOVL C00742 V=800.0 PL=0
MOVL C00743 V=800.0 PL=0
MOVL C00744 V=800.0 PL=0
MOVL C00745 V=800.0 PL=0
MOVL C00746 V=800.0 PL=0
MOVL C00747 V=800.0 PL=0
MOVL C00748 V=800.0 PL=0
MOVL C00749 V=800.0 PL=0
MOVL C00750 V=800.0 PL=0
MOVL C00751 V=800.0 PL=0
MOVL C00752 V=800.0 PL=0
MOVL C00753 V=800.0 PL=0
MOVL C00754 V=800.0 PL=0
MOVL C00755 V=800.0 PL=0
MOVL C00756 V=800.0 PL=0
MOVL C00757 V=800.0 PL=0
MOVL C00758 V=800.0 PL=0
MOVL C00759 V=800.0 PL=0
MOVL C00760 V=800.0 PL=0
MOVL C00761 V=800.0 PL=0
MOVL C00762 V=800.0 PL=0
MOVL C00763 V=800.0 PL=0
MOVL C00764 V=800.0 PL=0
MOVL C00765 V=800.0 PL=0
MOVL C00766 V=800.0 PL=0
MOVL C00767 V=800.0 PL=0
MOVL C00768 V=800.0 PL=0
MOVL C00769 V=800.0 PL=0
MOVL C00770 V=800.0 PL=0
MOVL C00771 V=800.0 PL=0
MOVL C00772 V=800.0 PL=0
MOVL C00773 V=800.0 PL=0
MOVL C00774 V=800.0 PL=0
MOVL C00775 V=800.0 PL=0
MOVL C00776 V=800.0 PL=0
MOVL C00777 V=800.0 PL=0
MOVL C00778 V=800.0 PL=0
MOVL C00779 V=800.0 PL=0
MOVL C00780 V=800.0 PL=0
MOVL C00781 V=800.0 PL=0
MOVL C00782 V=800.0 PL=0
MOVL C00783 V=800.0 PL=0
MOVL C00784 V=800.0 PL=0
MOVL C00785 V=800.0 PL=0
MOVL C00786 V=800.0 PL=0
MOVL C00787 V=800.0 PL=0
MOVL C00788 V=800.0 PL=0
MOVL C00789 V=800.0 PL=0
MOVL C00790 V=800.0 PL=0
MOVL C00791 V=800.0 PL=0
MOVL C00792 V=800.0 PL=0
MOVL C00793 V=800.0 PL=0
MOVL C00794 V=800.0 PL=0
MOVL C00795 V=800.0 PL=0
MOVL C00796 V=800.0 PL=0
MOVL C00797 V=800.0 PL=0
MOVL C00798 V=800.0 PL=0
MOVL C00799 V=800.0 PL=0
MOVL C00800 V=800.0 PL=0
MOVL C00801 V=800.0 PL=0
MOVL C00802 V=800.0 PL=0
MOVL C00803 V=800.0 PL=0
MOVL C00804 V=800.0 PL=0
MOVL C00805 V=800.0 PL=0
MOVL C00806 V=800.0 PL=0
MOVL C00807 V=800.0 PL=0
MOVL C00808 V=800.0 PL=0
MOVL C00809 V=800.0 PL=0
MOVL C00810 V=800.0 PL=0
MOVL C00811 V=800.0 PL=0
MOVL C00812 V=800.0 PL=0
MOVL C00813 V=800.0 PL=0
MOVL C00814 V=800.0 PL=0
MOVL C00815 V=800.0 PL=0
MOVL C00816 V=800.0 PL=0
MOVL C00817 V=800.0 PL=0
MOVL C00818 V=800.0 PL=0
MOVL C00819 V=800.0 PL=0
MOVL C00820 V=800.0 PL=0
MOVL C00821 V=800.0 PL=0
MOVL C00822 V=800.0 PL=0
MOVL C00823 V=800.0 PL=0
MOVL C00824 V=800.0 PL=0
MOVL C00825 V=800.0 PL=0
MOVL C00826 V=800.0 PL=0
MOVL C00827 V=800.0 PL=0
MOVL C00828 V=800.0 PL=0
MOVL C00829 V=800.0 PL=0
MOVL C00830 V=800.0 PL=0
MOVL C00831 V=800.0 PL=0
MOVL C00832 V=800.0 PL=0
MOVL C00833 V=800.0 PL=0
MOVL C00834 V=800.0 PL=0
MOVL C00835 V=800.0 PL=0
MOVL C00836 V=800.0 PL=0
MOVL C00837 V=800.0 PL=0
MOVL C00838 V=800.0 PL=0
MOVL C00839 V=800.0 PL=0
MOVL C00840 V=800.0 PL=0
MOVL C00841 V=800.0 PL=0
MOVL C00842 V=800.0 PL=0
MOVL C00843 V=800.0 PL=0
MOVL C00844 V=800.0 PL=0
MOVL C00845 V=800.0 PL=0
MOVL C00846 V=800.0 PL=0
MOVL C00847 V=800.0 PL=0
MOVL C00848 V=800.0 PL=0
MOVL C00849 V=800.0 PL=0
MOVL C00850 V=800.0 PL=0
MOVL C00851 V=800.0 PL=0
MOVL C00852 V=800.0 PL=0
MOVL C00853 V=800.0 PL=0
MOVL C00854 V=800.0 PL=0
MOVL C00855 V=800.0 PL=0
MOVL C00856 V=800.0 PL=0
MOVL C00857 V=800.0 PL=0
MOVL C00858 V=800.0 PL=0
MOVL C00859 V=800.0 PL=0
MOVL C00860 V=800.0 PL=0
MOVL C00861 V=800.0 PL=0
MOVL C00862 V=800.0 PL=0
MOVL C00863 V=800.0 PL=0
MOVL C00864 V=800.0 PL=0
MOVL C00865 V=800.0 PL=0
MOVL C00866 V=800.0 PL=0
MOVL C00867 V=800.0 PL=0
MOVL C00868 V=800.0 PL=0
MOVL C00869 V=800.0 PL=0
MOVL C00870 V=800.0 PL=0
MOVL C00871 V=800.0 PL=0
MOVL C00872 V=800.0 PL=0
MOVL C00873 V=800.0 PL=0
MOVL C00874 V=800.0 PL=0
MOVL C00875 V=800.0 PL=0
MOVL C00876 V=800.0 PL=0
MOVL C00877 V=800.0 PL=0
MOVL C00878 V=800.0 PL=0
MOVL C00879 V=800.0 PL=0
MOVL C00880 V=800.0 PL=0
MOVL C00881 V=800.0 PL=0
MOVL C00882 V=800.0 PL=0
MOVL C00883 V=800.0 PL=0
MOVL C00884 V=800.0 PL=0
MOVL C00885 V=800.0 PL=0
MOVL C00886 V=800.0 PL=0
MOVL C00887 V=800.0 PL=0
MOVL C00888 V=800.0 PL=0
MOVL C00889 V=800.0 PL=0
MOVL C00890 V=800.0 PL=0
MOVL C00891 V=800.0 PL=0
MOVL C00892 V=800.0 PL=0
MOVL C00893 V=800.0 PL=0
MOVL C00894 V=800.0 PL=0
MOVL C00895 V=800.0 PL=0
MOVL C00896 V=800.0 PL=0
MOVL C00897 V=800.0 PL=0
MOVL C00898 V=800.0 PL=0
MOVL C00899 V=800.0 PL=0
MOVL C00900 V=800.0 PL=0
MOVL C00901 V=800.0 PL=0
MOVL C00902 V=800.0 PL=0
MOVL C00903 V=800.0 PL=0
MOVL C00904 V=800.0 PL=0
MOVL C00905 V=800.0 PL=0
MOVL C00906 V=800.0 PL=0
MOVL C00907 V=800.0 PL=0
MOVL C00908 V=800.0 PL=0
MOVL C00909 V=800.0 PL=0
MOVL C00910 V=800.0 PL=0
MOVL C00911 V=800.0 PL=0
MOVL C00912 V=800.0 PL=0
MOVL C00913 V=800.0 PL=0
MOVL C00914 V=800.0 PL=0
MOVL C00915 V=800.0 PL=0
MOVL C00916 V=800.0 PL=0
MOVL C00917 V=800.0 PL=0
MOVL C00918 V=800.0 PL=0
MOVL C00919 V=800.0 PL=0
MOVL C00920 V=800.0 PL=0
MOVL C00921 V=800.0 PL=0
MOVL C00922 V=800.0 PL=0
MOVL C00923 V=800.0 PL=0
MOVL C00924 V=800.0 PL=0
MOVL C00925 V=800.0 PL=0
MOVL C00926 V=800.0 PL=0
MOVL C00927 V=800.0 PL=0
MOVL C00928 V=800.0 PL=0
MOVL C00929 V=800.0 PL=0
MOVL C00930 V=800.0 PL=0
MOVL C00931 V=800.0 PL=0
MOVL C00932 V=800.0 PL=0
MOVL C00933 V=800.0 PL=0
MOVL C00934 V=800.0 PL=0
MOVL C00935 V=800.0 PL=0
MOVL C00936 V=800.0 PL=0
MOVL C00937 V=800.0 PL=0
MOVL C00938 V=800.0 PL=0
MOVL C00939 V=800.0 PL=0
MOVL C00940 V=800.0 PL=0
MOVL C00941 V=800.0 PL=0
MOVL C00942 V=800.0 PL=0
MOVL C00943 V=800.0 PL=0
MOVL C00944 V=800.0 PL=0
MOVL C00945 V=800.0 PL=0
MOVL C00946 V=800.0 PL=0
MOVL C00947 V=800.0 PL=0
MOVL C00948 V=800.0 PL=0
MOVL C00949 V=800.0 PL=0
MOVL C00950 V=800.0 PL=0
MOVL C00951 V=800.0 PL=0
MOVL C00952 V=800.0 PL=0
MOVL C00953 V=800.0 PL=0
MOVL C00954 V=800.0 PL=0
MOVL C00955 V=800.0 PL=0
MOVL C00956 V=800.0 PL=0
MOVL C00957 V=800.0 PL=0
MOVL C00958 V=800.0 PL=0
MOVL C00959 V=800.0 PL=0
MOVL C00960 V=800.0 PL=0
MOVL C00961 V=800.0 PL=0
MOVL C00962 V=800.0 PL=0
MOVL C00963 V=800.0 PL=0
MOVL C00964 V=800.0 PL=0
MOVL C00965 V=800.0 PL=0
MOVL C00966 V=800.0 PL=0
MOVL C00967 V=800.0 PL=0
MOVL C00968 V=800.0 PL=0
MOVL C00969 V=800.0 PL=0
MOVL C00970 V=800.0 PL=0
MOVL C00971 V=800.0 PL=0
MOVL C00972 V=800.0 PL=0
MOVL C00973 V=800.0 PL=0
MOVL C00974 V=800.0 PL=0
MOVL C00975 V=800.0 PL=0
MOVL C00976 V=800.0 PL=0
MOVL C00977 V=800.0 PL=0
MOVL C00978 V=800.0 PL=0
MOVL C00979 V=800.0 PL=0
MOVL C00980 V=800.0 PL=0
MOVL C00981 V=800.0 PL=0
MOVL C00982 V=800.0 PL=0
MOVL C00983 V=800.0 PL=0
MOVL C00984 V=800.0 PL=0
MOVL C00985 V=800.0 PL=0
MOVL C00986 V=800.0 PL=0
MOVL C00987 V=800.0 PL=0
MOVL C00988 V=800.0 PL=0
MOVL C00989 V=800.0 PL=0
MOVL C00990 V=800.0 PL=0
MOVL C00991 V=800.0 PL=0
MOVL C00992 V=800.0 PL=0
MOVL C00993 V=800.0 PL=0
MOVL C00994 V=800.0 PL=0
MOVL C00995 V=800.0 PL=0
MOVL C00996 V=800.0 PL=0
MOVL C00997 V=800.0 PL=0
MOVL C00998 V=800.0 PL=0
MOVL C00999 V=800.0 PL=0
MOVL C01000 V=800.0 PL=0
MOVL C01001 V=800.0 PL=0
MOVL C01002 V=800.0 PL=0
MOVL C01003 V=800.0 PL=0
MOVL C01004 V=800.0 PL=0
MOVL C01005 V=800.0 PL=0
MOVL C01006 V=800.0 PL=0
MOVL C01007 V=800.0 PL=0
MOVL C01008 V=800.0 PL=0
MOVL C01009 V=800.0 PL=0
MOVL C01010 V=800.0 PL=0
MOVL C01011 V=800.0 PL=0
MOVL C01012 V=800.0 PL=0
MOVL C01013 V=800.0 PL=0
MOVL C01014 V=800.0 PL=0
MOVL C01015 V=800.0 PL=0
MOVL C01016 V=800.0 PL=0
MOVL C01017 V=800.0 PL=0
MOVL C01018 V=800.0 PL=0
MOVL C01019 V=800.0 PL=0
MOVL C01020 V=800.0 PL=0
MOVL C01021 V=800.0 PL=0
MOVL C01022 V=800.0 PL=0
MOVL C01023 V=800.0 PL=0
MOVL C01024 V=800.0 PL=0
MOVL C01025 V=800.0 PL=0
MOVL C01026 V=800.0 PL=0
MOVL C01027 V=800.0 PL=0
MOVL C01028 V=800.0 PL=0
MOVL C01029 V=800.0 PL=0
MOVL C01030 V=800.0 PL=0
MOVL C01031 V=800.0 PL=0
MOVL C01032 V=800.0 PL=0
MOVL C01033 V=800.0 PL=0
MOVL C01034 V=800.0 PL=0
MOVL C01035 V=800.0 PL=0
MOVL C01036 V=800.0 PL=0
MOVL C01037 V=800.0 PL=0
MOVL C01038 V=800.0 PL=0
MOVL C01039 V=800.0 PL=0
MOVL C01040 V=800.0 PL=0
MOVL C01041 V=800.0 PL=0
MOVL C01042 V=800.0 PL=0
MOVL C01043 V=800.0 PL=0
MOVL C01044 V=800.0 PL=0
MOVL C01045 V=800.0 PL=0
MOVL C01046 V=800.0 PL=0
MOVL C01047 V=800.0 PL=0
MOVL C01048 V=800.0 PL=0
MOVL C01049 V=800.0 PL=0
MOVL C01050 V=800.0 PL=0
MOVL C01051 V=800.0 PL=0
MOVL C01052 V=800.0 PL=0
MOVL C01053 V=800.0 PL=0
MOVL C01054 V=800.0 PL=0
MOVL C01055 V=800.0 PL=0
MOVL C01056 V=800.0 PL=0
MOVL C01057 V=800.0 PL=0
MOVL C01058 V=800.0 PL=0
MOVL C01059 V=800.0 PL=0
MOVL C01060 V=800.0 PL=0
MOVL C01061 V=800.0 PL=0
MOVL C01062 V=800.0 PL=0
MOVL C01063 V=800.0 PL=0
MOVL C01064 V=800.0 PL=0
MOVL C01065 V=800.0 PL=0
MOVL C01066 V=800.0 PL=0
MOVL C01067 V=800.0 PL=0
MOVL C01068 V=800.0 PL=0
MOVL C01069 V=800.0 PL=0
MOVL C01070 V=800.0 PL=0
MOVL C01071 V=800.0 PL=0
MOVL C01072 V=800.0 PL=0
MOVL C01073 V=800.0 PL=0
MOVL C01074 V=800.0 PL=0
MOVL C01075 V=800.0 PL=0
MOVL C01076 V=800.0 PL=0
MOVL C01077 V=800.0 PL=0
MOVL C01078 V=800.0 PL=0
MOVL C01079 V=800.0 PL=0
MOVL C01080 V=800.0 PL=0
MOVL C01081 V=800.0 PL=0
MOVL C01082 V=800.0 PL=0
MOVL C01083 V=800.0 PL=0
MOVL C01084 V=800.0 PL=0
MOVL C01085 V=800.0 PL=0
MOVL C01086 V=800.0 PL=0
MOVL C01087 V=800.0 PL=0
MOVL C01088 V=800.0 PL=0
MOVL C01089 V=800.0 PL=0
MOVL C01090 V=800.0 PL=0
MOVL C01091 V=800.0 PL=0
MOVL C01092 V=800.0 PL=0
MOVL C01093 V=800.0 PL=0
MOVL C01094 V=800.0 PL=0
MOVL C01095 V=800.0 PL=0
MOVL C01096 V=800.0 PL=0
MOVL C01097 V=800.0 PL=0
MOVL C01098 V=800.0 PL=0
MOVL C01099 V=800.0 PL=0
MOVL C01100 V=800.0 PL=0
MOVL C01101 V=800.0 PL=0
MOVL C01102 V=800.0 PL=0
MOVL C01103 V=800.0 PL=0
MOVL C01104 V=800.0 PL=0
MOVL C01105 V=800.0 PL=0
MOVL C01106 V=800.0 PL=0
MOVL C01107 V=800.0 PL=0
MOVL C01108 V=800.0 PL=0
MOVL C01109 V=800.0 PL=0
MOVL C01110 V=800.0 PL=0
MOVL C01111 V=800.0 PL=0
MOVL C01112 V=800.0 PL=0
MOVL C01113 V=800.0 PL=0
MOVL C01114 V=800.0 PL=0
MOVL C01115 V=800.0 PL=0
MOVL C01116 V=800.0 PL=0
MOVL C01117 V=800.0 PL=0
MOVL C01118 V=800.0 PL=0
MOVL C01119 V=800.0 PL=0
MOVL C01120 V=800.0 PL=0
MOVL C01121 V=800.0 PL=0
MOVL C01122 V=800.0 PL=0
MOVL C01123 V=800.0 PL=0
MOVL C01124 V=800.0 PL=0
MOVL C01125 V=800.0 PL=0
MOVL C01126 V=800.0 PL=0
MOVL C01127 V=800.0 PL=0
MOVL C01128 V=800.0 PL=0
MOVL C01129 V=800.0 PL=0
MOVL C01130 V=800.0 PL=0
MOVL C01131 V=800.0 PL=0
MOVL C01132 V=800.0 PL=0
MOVL C01133 V=800.0 PL=0
MOVL C01134 V=800.0 PL=0
MOVL C01135 V=800.0 PL=0
MOVL C01136 V=800.0 PL=0
MOVL C01137 V=800.0 PL=0
MOVL C01138 V=800.0 PL=0
MOVL C01139 V=800.0 PL=0
MOVL C01140 V=800.0 PL=0
MOVL C01141 V=800.0 PL=0
MOVL C01142 V=800.0 PL=0
MOVL C01143 V=800.0 PL=0
MOVL C01144 V=800.0 PL=0
MOVL C01145 V=800.0 PL=0
MOVL C01146 V=800.0 PL=0
MOVL C01147 V=800.0 PL=0
MOVL C01148 V=800.0 PL=0
MOVL C01149 V=800.0 PL=0
MOVL C01150 V=800.0 PL=0
MOVL C01151 V=800.0 PL=0
MOVL C01152 V=800.0 PL=0
MOVL C01153 V=800.0 PL=0
MOVL C01154 V=800.0 PL=0
MOVL C01155 V=800.0 PL=0
MOVL C01156 V=800.0 PL=0
MOVL C01157 V=800.0 PL=0
MOVL C01158 V=800.0 PL=0
MOVL C01159 V=800.0 PL=0
MOVL C01160 V=800.0 PL=0
MOVL C01161 V=800.0 PL=0
MOVL C01162 V=800.0 PL=0
MOVL C01163 V=800.0 PL=0
MOVL C01164 V=800.0 PL=0
MOVL C01165 V=800.0 PL=0
MOVL C01166 V=800.0 PL=0
MOVL C01167 V=800.0 PL=0
MOVL C01168 V=800.0 PL=0
MOVL C01169 V=800.0 PL=0
MOVL C01170 V=800.0 PL=0
MOVL C01171 V=800.0 PL=0
MOVL C01172 V=800.0 PL=0
MOVL C01173 V=800.0 PL=0
MOVL C01174 V=800.0 PL=0
MOVL C01175 V=800.0 PL=0
MOVL C01176 V=800.0 PL=0
MOVL C01177 V=800.0 PL=0
MOVL C01178 V=800.0 PL=0
MOVL C01179 V=800.0 PL=0
MOVL C01180 V=800.0 PL=0
MOVL C01181 V=800.0 PL=0
MOVL C01182 V=800.0 PL=0
MOVL C01183 V=800.0 PL=0
MOVL C01184 V=800.0 PL=0
MOVL C01185 V=800.0 PL=0
MOVL C01186 V=800.0 PL=0
MOVL C01187 V=800.0 PL=0
MOVL C01188 V=800.0 PL=0
MOVL C01189 V=800.0 PL=0
MOVL C01190 V=800.0 PL=0
MOVL C01191 V=800.0 PL=0
MOVL C01192 V=800.0 PL=0
MOVL C01193 V=800.0 PL=0
MOVL C01194 V=800.0 PL=0
MOVL C01195 V=800.0 PL=0
MOVL C01196 V=800.0 PL=0
MOVL C01197 V=800.0 PL=0
MOVL C01198 V=800.0 PL=0
MOVL C01199 V=800.0 PL=0
MOVL C01200 V=800.0 PL=0
MOVL C01201 V=800.0 PL=0
MOVL C01202 V=800.0 PL=0
MOVL C01203 V=800.0 PL=0
MOVL C01204 V=800.0 PL=0
MOVL C01205 V=800.0 PL=0
MOVL C01206 V=800.0 PL=0
MOVL C01207 V=800.0 PL=0
MOVL C01208 V=800.0 PL=0
MOVL C01209 V=800.0 PL=0
MOVL C01210 V=800.0 PL=0
MOVL C01211 V=800.0 PL=0
MOVL C01212 V=800.0 PL=0
MOVL C01213 V=800.0 PL=0
MOVL C01214 V=800.0 PL=0
MOVL C01215 V=800.0 PL=0
MOVL C01216 V=800.0 PL=0
MOVL C01217 V=800.0 PL=0
MOVL C01218 V=800.0 PL=0
MOVL C01219 V=800.0 PL=0
MOVL C01220 V=800.0 PL=0
MOVL C01221 V=800.0 PL=0
MOVL C01222 V=800.0 PL=0
MOVL C01223 V=800.0 PL=0
MOVL C01224 V=800.0 PL=0
MOVL C01225 V=800.0 PL=0
MOVL C01226 V=800.0 PL=0
MOVL C01227 V=800.0 PL=0
MOVL C01228 V=800.0 PL=0
MOVL C01229 V=800.0 PL=0
MOVL C01230 V=800.0 PL=0
MOVL C01231 V=800.0 PL=0
MOVL C01232 V=800.0 PL=0
MOVL C01233 V=800.0 PL=0
MOVL C01234 V=800.0 PL=0
MOVL C01235 V=800.0 PL=0
MOVL C01236 V=800.0 PL=0
MOVL C01237 V=800.0 PL=0
MOVL C01238 V=800.0 PL=0
MOVL C01239 V=800.0 PL=0
MOVL C01240 V=800.0 PL=0
MOVL C01241 V=800.0 PL=0
MOVL C01242 V=800.0 PL=0
MOVL C01243 V=800.0 PL=0
MOVL C01244 V=800.0 PL=0
MOVL C01245 V=800.0 PL=0
MOVL C01246 V=800.0 PL=0
MOVL C01247 V=800.0 PL=0
MOVL C01248 V=800.0 PL=0
MOVL C01249 V=800.0 PL=0
MOVL C01250 V=800.0 PL=0
MOVL C01251 V=800.0 PL=0
MOVL C01252 V=800.0 PL=0
MOVL C01253 V=800.0 PL=0
MOVL C01254 V=800.0 PL=0
MOVL C01255 V=800.0 PL=0
MOVL C01256 V=800.0 PL=0
MOVL C01257 V=800.0 PL=0
MOVL C01258 V=800.0 PL=0
MOVL C01259 V=800.0 PL=0
MOVL C01260 V=800.0 PL=0
MOVL C01261 V=800.0 PL=0
MOVL C01262 V=800.0 PL=0
MOVL C01263 V=800.0 PL=0
MOVL C01264 V=800.0 PL=0
MOVL C01265 V=800.0 PL=0
MOVL C01266 V=800.0 PL=0
MOVL C01267 V=800.0 PL=0
MOVL C01268 V=800.0 PL=0
MOVL C01269 V=800.0 PL=0
MOVL C01270 V=800.0 PL=0
MOVL C01271 V=800.0 PL=0
MOVL C01272 V=800.0 PL=0
MOVL C01273 V=800.0 PL=0
MOVL C01274 V=800.0 PL=0
MOVL C01275 V=800.0 PL=0
MOVL C01276 V=800.0 PL=0
MOVL C01277 V=800.0 PL=0
MOVL C01278 V=800.0 PL=0
MOVL C01279 V=800.0 PL=0
MOVL C01280 V=800.0 PL=0
MOVL C01281 V=800.0 PL=0
MOVL C01282 V=800.0 PL=0
MOVL C01283 V=800.0 PL=0
MOVL C01284 V=800.0 PL=0
MOVL C01285 V=800.0 PL=0
MOVL C01286 V=800.0 PL=0
MOVL C01287 V=800.0 PL=0
MOVL C01288 V=800.0 PL=0
MOVL C01289 V=800.0 PL=0
MOVL C01290 V=800.0 PL=0
MOVL C01291 V=800.0 PL=0
MOVL C01292 V=800.0 PL=0
MOVL C01293 V=800.0 PL=0
MOVL C01294 V=800.0 PL=0
MOVL C01295 V=800.0 PL=0
MOVL C01296 V=800.0 PL=0
MOVL C01297 V=800.0 PL=0
MOVL C01298 V=800.0 PL=0
MOVL C01299 V=800.0 PL=0
MOVL C01300 V=800.0 PL=0
MOVL C01301 V=800.0 PL=0
MOVL C01302 V=800.0 PL=0
MOVL C01303 V=800.0 PL=0
MOVL C01304 V=800.0 PL=0
MOVL C01305 V=800.0 PL=0
MOVL C01306 V=800.0 PL=0
MOVL C01307 V=800.0 PL=0
MOVL C01308 V=800.0 PL=0
MOVL C01309 V=800.0 PL=0
MOVL C01310 V=800.0 PL=0
MOVL C01311 V=800.0 PL=0
MOVL C01312 V=800.0 PL=0
MOVL C01313 V=800.0 PL=0
MOVL C01314 V=800.0 PL=0
MOVL C01315 V=800.0 PL=0
MOVL C01316 V=800.0 PL=0
MOVL C01317 V=800.0 PL=0
MOVL C01318 V=800.0 PL=0
MOVL C01319 V=800.0 PL=0
MOVL C01320 V=800.0 PL=0
MOVL C01321 V=800.0 PL=0
MOVL C01322 V=800.0 PL=0
MOVL C01323 V=800.0 PL=0
MOVL C01324 V=800.0 PL=0
MOVL C01325 V=800.0 PL=0
MOVL C01326 V=800.0 PL=0
MOVL C01327 V=800.0 PL=0
MOVL C01328 V=800.0 PL=0
MOVL C01329 V=800.0 PL=0
MOVL C01330 V=800.0 PL=0
MOVL C01331 V=800.0 PL=0
MOVL C01332 V=800.0 PL=0
MOVL C01333 V=800.0 PL=0
MOVL C01334 V=800.0 PL=0
MOVL C01335 V=800.0 PL=0
MOVL C01336 V=800.0 PL=0
MOVL C01337 V=800.0 PL=0
MOVL C01338 V=800.0 PL=0
MOVL C01339 V=800.0 PL=0
MOVL C01340 V=800.0 PL=0
MOVL C01341 V=800.0 PL=0
MOVL C01342 V=800.0 PL=0
MOVL C01343 V=800.0 PL=0
MOVL C01344 V=800.0 PL=0
MOVL C01345 V=800.0 PL=0
MOVL C01346 V=800.0 PL=0
MOVL C01347 V=800.0 PL=0
MOVL C01348 V=800.0 PL=0
MOVL C01349 V=800.0 PL=0
MOVL C01350 V=800.0 PL=0
MOVL C01351 V=800.0 PL=0
MOVL C01352 V=800.0 PL=0
MOVL C01353 V=800.0 PL=0
MOVL C01354 V=800.0 PL=0
MOVL C01355 V=800.0 PL=0
MOVL C01356 V=800.0 PL=0
MOVL C01357 V=800.0 PL=0
MOVL C01358 V=800.0 PL=0
MOVL C01359 V=800.0 PL=0
MOVL C01360 V=800.0 PL=0
MOVL C01361 V=800.0 PL=0
MOVL C01362 V=800.0 PL=0
MOVL C01363 V=800.0 PL=0
MOVL C01364 V=800.0 PL=0
MOVL C01365 V=800.0 PL=0
MOVL C01366 V=800.0 PL=0
MOVL C01367 V=800.0 PL=0
MOVL C01368 V=800.0 PL=0
MOVL C01369 V=800.0 PL=0
MOVL C01370 V=800.0 PL=0
MOVL C01371 V=800.0 PL=0
MOVL C01372 V=800.0 PL=0
MOVL C01373 V=800.0 PL=0
MOVL C01374 V=800.0 PL=0
MOVL C01375 V=800.0 PL=0
MOVL C01376 V=800.0 PL=0
MOVL C01377 V=800.0 PL=0
MOVL C01378 V=800.0 PL=0
MOVL C01379 V=800.0 PL=0
MOVL C01380 V=800.0 PL=0
MOVL C01381 V=800.0 PL=0
MOVL C01382 V=800.0 PL=0
MOVL C01383 V=800.0 PL=0
MOVL C01384 V=800.0 PL=0
MOVL C01385 V=800.0 PL=0
MOVL C01386 V=800.0 PL=0
MOVL C01387 V=800.0 PL=0
MOVL C01388 V=800.0 PL=0
MOVL C01389 V=800.0 PL=0
MOVL C01390 V=800.0 PL=0
MOVL C01391 V=800.0 PL=0
MOVL C01392 V=800.0 PL=0
MOVL C01393 V=800.0 PL=0
MOVL C01394 V=800.0 PL=0
MOVL C01395 V=800.0 PL=0
MOVL C01396 V=800.0 PL=0
MOVL C01397 V=800.0 PL=0
MOVL C01398 V=800.0 PL=0
MOVL C01399 V=800.0 PL=0
MOVL C01400 V=800.0 PL=0
MOVL C01401 V=800.0 PL=0
MOVL C01402 V=800.0 PL=0
MOVL C01403 V=800.0 PL=0
MOVL C01404 V=800.0 PL=0
MOVL C01405 V=800.0 PL=0
MOVL C01406 V=800.0 PL=0
MOVL C01407 V=800.0 PL=0
MOVL C01408 V=800.0 PL=0
MOVL C01409 V=800.0 PL=0
MOVL C01410 V=800.0 PL=0
MOVL C01411 V=800.0 PL=0
MOVL C01412 V=800.0 PL=0
MOVL C01413 V=800.0 PL=0
MOVL C01414 V=800.0 PL=0
MOVL C01415 V=800.0 PL=0
MOVL C01416 V=800.0 PL=0
MOVL C01417 V=800.0 PL=0
MOVL C01418 V=800.0 PL=0
MOVL C01419 V=800.0 PL=0
MOVL C01420 V=800.0 PL=0
MOVL C01421 V=800.0 PL=0
MOVL C01422 V=800.0 PL=0
MOVL C01423 V=800.0 PL=0
MOVL C01424 V=800.0 PL=0
MOVL C01425 V=800.0 PL=0
MOVL C01426 V=800.0 PL=0
MOVL C01427 V=800.0 PL=0
MOVL C01428 V=800.0 PL=0
MOVL C01429 V=800.0 PL=0
MOVL C01430 V=800.0 PL=0
MOVL C01431 V=800.0 PL=0
MOVL C01432 V=800.0 PL=0
MOVL C01433 V=800.0 PL=0
MOVL C01434 V=800.0 PL=0
MOVL C01435 V=800.0 PL=0
MOVL C01436 V=800.0 PL=0
MOVL C01437 V=800.0 PL=0
MOVL C01438 V=800.0 PL=0
MOVL C01439 V=800.0 PL=0
MOVL C01440 V=800.0 PL=0
MOVL C01441 V=800.0 PL=0
MOVL C01442 V=800.0 PL=0
MOVL C01443 V=800.0 PL=0
MOVL C01444 V=800.0 PL=0
MOVL C01445 V=800.0 PL=0
MOVL C01446 V=800.0 PL=0
MOVL C01447 V=800.0 PL=0
MOVL C01448 V=800.0 PL=0
MOVL C01449 V=800.0 PL=0
MOVL C01450 V=800.0 PL=0
MOVL C01451 V=800.0 PL=0
MOVL C01452 V=800.0 PL=0
MOVL C01453 V=800.0 PL=0
MOVL C01454 V=800.0 PL=0
MOVL C01455 V=800.0 PL=0
MOVL C01456 V=800.0 PL=0
MOVL C01457 V=800.0 PL=0
MOVL C01458 V=800.0 PL=0
MOVL C01459 V=800.0 PL=0
MOVL C01460 V=800.0 PL=0
MOVL C01461 V=800.0 PL=0
MOVL C01462 V=800.0 PL=0
MOVL C01463 V=800.0 PL=0
MOVL C01464 V=800.0 PL=0
MOVL C01465 V=800.0 PL=0
MOVL C01466 V=800.0 PL=0
MOVL C01467 V=800.0 PL=0
MOVL C01468 V=800.0 PL=0
MOVL C01469 V=800.0 PL=0
MOVL C01470 V=800.0 PL=0
MOVL C01471 V=800.0 PL=0
MOVL C01472 V=800.0 PL=0
MOVL C01473 V=800.0 PL=0
MOVL C01474 V=800.0 PL=0
MOVL C01475 V=800.0 PL=0
MOVL C01476 V=800.0 PL=0
MOVL C01477 V=800.0 PL=0
MOVL C01478 V=800.0 PL=0
MOVL C01479 V=800.0 PL=0
MOVL C01480 V=800.0 PL=0
MOVL C01481 V=800.0 PL=0
MOVL C01482 V=800.0 PL=0
MOVL C01483 V=800.0 PL=0
MOVL C01484 V=800.0 PL=0
MOVL C01485 V=800.0 PL=0
MOVL C01486 V=800.0 PL=0
MOVL C01487 V=800.0 PL=0
MOVL C01488 V=800.0 PL=0
MOVL C01489 V=800.0 PL=0
MOVL C01490 V=800.0 PL=0
MOVL C01491 V=800.0 PL=0
MOVL C01492 V=800.0 PL=0
MOVL C01493 V=800.0 PL=0
MOVL C01494 V=800.0 PL=0
MOVL C01495 V=800.0 PL=0
MOVL C01496 V=800.0 PL=0
MOVL C01497 V=800.0 PL=0
MOVL C01498 V=800.0 PL=0
MOVL C01499 V=800.0 PL=0
MOVL C01500 V=800.0 PL=0
MOVL C01501 V=800.0 PL=0
MOVL C01502 V=800.0 PL=0
MOVL C01503 V=800.0 PL=0
MOVL C01504 V=800.0 PL=0
MOVL C01505 V=800.0 PL=0
MOVL C01506 V=800.0 PL=0
MOVL C01507 V=800.0 PL=0
MOVL C01508 V=800.0 PL=0
MOVL C01509 V=800.0 PL=0
MOVL C01510 V=800.0 PL=0
MOVL C01511 V=800.0 PL=0
MOVL C01512 V=800.0 PL=0
MOVL C01513 V=800.0 PL=0
MOVL C01514 V=800.0 PL=0
MOVL C01515 V=800.0 PL=0
MOVL C01516 V=800.0 PL=0
MOVL C01517 V=800.0 PL=0
MOVL C01518 V=800.0 PL=0
MOVL C01519 V=800.0 PL=0
MOVL C01520 V=800.0 PL=0
MOVL C01521 V=800.0 PL=0
MOVL C01522 V=800.0 PL=0
MOVL C01523 V=800.0 PL=0
MOVL C01524 V=800.0 PL=0
MOVL C01525 V=800.0 PL=0
MOVL C01526 V=800.0 PL=0
MOVL C01527 V=800.0 PL=0
MOVL C01528 V=800.0 PL=0
MOVL C01529 V=800.0 PL=0
MOVL C01530 V=800.0 PL=0
MOVL C01531 V=800.0 PL=0
MOVL C01532 V=800.0 PL=0
MOVL C01533 V=800.0 PL=0
MOVL C01534 V=800.0 PL=0
MOVL C01535 V=800.0 PL=0
MOVL C01536 V=800.0 PL=0
MOVL C01537 V=800.0 PL=0
MOVL C01538 V=800.0 PL=0
MOVL C01539 V=800.0 PL=0
MOVL C01540 V=800.0 PL=0
MOVL C01541 V=800.0 PL=0
MOVL C01542 V=800.0 PL=0
MOVL C01543 V=800.0 PL=0
MOVL C01544 V=800.0 PL=0
MOVL C01545 V=800.0 PL=0
MOVL C01546 V=800.0 PL=0
MOVL C01547 V=800.0 PL=0
MOVL C01548 V=800.0 PL=0
MOVL C01549 V=800.0 PL=0
MOVL C01550 V=800.0 PL=0
MOVL C01551 V=800.0 PL=0
MOVL C01552 V=800.0 PL=0
MOVL C01553 V=800.0 PL=0
MOVL C01554 V=800.0 PL=0
MOVL C01555 V=800.0 PL=0
MOVL C01556 V=800.0 PL=0
MOVL C01557 V=800.0 PL=0
MOVL C01558 V=800.0 PL=0
MOVL C01559 V=800.0 PL=0
MOVL C01560 V=800.0 PL=0
MOVL C01561 V=800.0 PL=0
MOVL C01562 V=800.0 PL=0
MOVL C01563 V=800.0 PL=0
MOVL C01564 V=800.0 PL=0
MOVL C01565 V=800.0 PL=0
MOVL C01566 V=800.0 PL=0
MOVL C01567 V=800.0 PL=0
MOVL C01568 V=800.0 PL=0
MOVL C01569 V=800.0 PL=0
MOVL C01570 V=800.0 PL=0
MOVL C01571 V=800.0 PL=0
MOVL C01572 V=800.0 PL=0
MOVL C01573 V=800.0 PL=0
MOVL C01574 V=800.0 PL=0
MOVL C01575 V=800.0 PL=0
MOVL C01576 V=800.0 PL=0
MOVL C01577 V=800.0 PL=0
MOVL C01578 V=800.0 PL=0
MOVL C01579 V=800.0 PL=0
MOVL C01580 V=800.0 PL=0
MOVL C01581 V=800.0 PL=0
MOVL C01582 V=800.0 PL=0
MOVL C01583 V=800.0 PL=0
MOVL C01584 V=800.0 PL=0
MOVL C01585 V=800.0 PL=0
MOVL C01586 V=800.0 PL=0
MOVL C01587 V=800.0 PL=0
MOVL C01588 V=800.0 PL=0
MOVL C01589 V=800.0 PL=0
MOVL C01590 V=800.0 PL=0
MOVL C01591 V=800.0 PL=0
MOVL C01592 V=800.0 PL=0
MOVL C01593 V=800.0 PL=0
MOVL C01594 V=800.0 PL=0
MOVL C01595 V=800.0 PL=0
MOVL C01596 V=800.0 PL=0
MOVL C01597 V=800.0 PL=0
MOVL C01598 V=800.0 PL=0
MOVL C01599 V=800.0 PL=0
MOVL C01600 V=800.0 PL=0
MOVL C01601 V=800.0 PL=0
MOVL C01602 V=800.0 PL=0
MOVL C01603 V=800.0 PL=0
MOVL C01604 V=800.0 PL=0
MOVL C01605 V=800.0 PL=0
MOVL C01606 V=800.0 PL=0
MOVL C01607 V=800.0 PL=0
MOVL C01608 V=800.0 PL=0
MOVL C01609 V=800.0 PL=0
MOVL C01610 V=800.0 PL=0
MOVL C01611 V=800.0 PL=0
MOVL C01612 V=800.0 PL=0
MOVL C01613 V=800.0 PL=0
MOVL C01614 V=800.0 PL=0
MOVL C01615 V=800.0 PL=0
MOVL C01616 V=800.0 PL=0
MOVL C01617 V=800.0 PL=0
MOVL C01618 V=800.0 PL=0
MOVL C01619 V=800.0 PL=0
MOVL C01620 V=800.0 PL=0
MOVL C01621 V=800.0 PL=0
MOVL C01622 V=800.0 PL=0
MOVL C01623 V=800.0 PL=0
MOVL C01624 V=800.0 PL=0
MOVL C01625 V=800.0 PL=0
MOVL C01626 V=800.0 PL=0
MOVL C01627 V=800.0 PL=0
MOVL C01628 V=800.0 PL=0
MOVL C01629 V=800.0 PL=0
MOVL C01630 V=800.0 PL=0
MOVL C01631 V=800.0 PL=0
MOVL C01632 V=800.0 PL=0
MOVL C01633 V=800.0 PL=0
MOVL C01634 V=800.0 PL=0
MOVL C01635 V=800.0 PL=0
MOVL C01636 V=800.0 PL=0
MOVL C01637 V=800.0 PL=0
MOVL C01638 V=800.0 PL=0
MOVL C01639 V=800.0 PL=0
MOVL C01640 V=800.0 PL=0
MOVL C01641 V=800.0 PL=0
MOVL C01642 V=800.0 PL=0
MOVL C01643 V=800.0 PL=0
MOVL C01644 V=800.0 PL=0
MOVL C01645 V=800.0 PL=0
MOVL C01646 V=800.0 PL=0
MOVL C01647 V=800.0 PL=0
MOVL C01648 V=800.0 PL=0
MOVL C01649 V=800.0 PL=0
MOVL C01650 V=800.0 PL=0
MOVL C01651 V=800.0 PL=0
MOVL C01652 V=800.0 PL=0
MOVL C01653 V=800.0 PL=0
MOVL C01654 V=800.0 PL=0
MOVL C01655 V=800.0 PL=0
MOVL C01656 V=800.0 PL=0
MOVL C01657 V=800.0 PL=0
MOVL C01658 V=800.0 PL=0
MOVL C01659 V=800.0 PL=0
MOVL C01660 V=800.0 PL=0
MOVL C01661 V=800.0 PL=0
MOVL C01662 V=800.0 PL=0
MOVL C01663 V=800.0 PL=0
MOVL C01664 V=800.0 PL=0
MOVL C01665 V=800.0 PL=0
MOVL C01666 V=800.0 PL=0
MOVL C01667 V=800.0 PL=0
MOVL C01668 V=800.0 PL=0
MOVL C01669 V=800.0 PL=0
MOVL C01670 V=800.0 PL=0
MOVL C01671 V=800.0 PL=0
MOVL C01672 V=800.0 PL=0
MOVL C01673 V=800.0 PL=0
MOVL C01674 V=800.0 PL=0
MOVL C01675 V=800.0 PL=0
MOVL C01676 V=800.0 PL=0
MOVL C01677 V=800.0 PL=0
MOVL C01678 V=800.0 PL=0
MOVL C01679 V=800.0 PL=0
MOVL C01680 V=800.0 PL=0
MOVL C01681 V=800.0 PL=0
MOVL C01682 V=800.0 PL=0
MOVL C01683 V=800.0 PL=0
MOVL C01684 V=800.0 PL=0
MOVL C01685 V=800.0 PL=0
MOVL C01686 V=800.0 PL=0
MOVL C01687 V=800.0 PL=0
MOVL C01688 V=800.0 PL=0
MOVL C01689 V=800.0 PL=0
MOVL C01690 V=800.0 PL=0
MOVL C01691 V=800.0 PL=0
MOVL C01692 V=800.0 PL=0
MOVL C01693 V=800.0 PL=0
MOVL C01694 V=800.0 PL=0
MOVL C01695 V=800.0 PL=0
MOVL C01696 V=800.0 PL=0
MOVL C01697 V=800.0 PL=0
MOVL C01698 V=800.0 PL=0
MOVL C01699 V=800.0 PL=0
MOVL C01700 V=800.0 PL=0
MOVL C01701 V=800.0 PL=0
MOVL C01702 V=800.0 PL=0
MOVL C01703 V=800.0 PL=0
MOVL C01704 V=800.0 PL=0
MOVL C01705 V=800.0 PL=0
MOVL C01706 V=800.0 PL=0
MOVL C01707 V=800.0 PL=0
MOVL C01708 V=800.0 PL=0
MOVL C01709 V=800.0 PL=0
MOVL C01710 V=800.0 PL=0
MOVL C01711 V=800.0 PL=0
MOVL C01712 V=800.0 PL=0
MOVL C01713 V=800.0 PL=0
MOVL C01714 V=800.0 PL=0
MOVL C01715 V=800.0 PL=0
MOVL C01716 V=800.0 PL=0
MOVL C01717 V=800.0 PL=0
MOVL C01718 V=800.0 PL=0
MOVL C01719 V=800.0 PL=0
MOVL C01720 V=800.0 PL=0
MOVL C01721 V=800.0 PL=0
MOVL C01722 V=800.0 PL=0
MOVL C01723 V=800.0 PL=0
MOVL C01724 V=800.0 PL=0
MOVL C01725 V=800.0 PL=0
MOVL C01726 V=800.0 PL=0
MOVL C01727 V=800.0 PL=0
MOVL C01728 V=800.0 PL=0
MOVL C01729 V=800.0 PL=0
MOVL C01730 V=800.0 PL=0
MOVL C01731 V=800.0 PL=0
MOVL C01732 V=800.0 PL=0
MOVL C01733 V=800.0 PL=0
MOVL C01734 V=800.0 PL=0
MOVL C01735 V=800.0 PL=0
MOVL C01736 V=800.0 PL=0
MOVL C01737 V=800.0 PL=0
MOVL C01738 V=800.0 PL=0
MOVL C01739 V=800.0 PL=0
MOVL C01740 V=800.0 PL=0
MOVL C01741 V=800.0 PL=0
MOVL C01742 V=800.0 PL=0
MOVL C01743 V=800.0 PL=0
MOVL C01744 V=800.0 PL=0
MOVL C01745 V=800.0 PL=0
MOVL C01746 V=800.0 PL=0
MOVL C01747 V=800.0 PL=0
MOVL C01748 V=800.0 PL=0
MOVL C01749 V=800.0 PL=0
MOVL C01750 V=800.0 PL=0
MOVL C01751 V=800.0 PL=0
MOVL C01752 V=800.0 PL=0
MOVL C01753 V=800.0 PL=0
MOVL C01754 V=800.0 PL=0
MOVL C01755 V=800.0 PL=0
MOVL C01756 V=800.0 PL=0
MOVL C01757 V=800.0 PL=0
MOVL C01758 V=800.0 PL=0
MOVL C01759 V=800.0 PL=0
MOVL C01760 V=800.0 PL=0
MOVL C01761 V=800.0 PL=0
MOVL C01762 V=800.0 PL=0
MOVL C01763 V=800.0 PL=0
MOVL C01764 V=800.0 PL=0
MOVL C01765 V=800.0 PL=0
MOVL C01766 V=800.0 PL=0
MOVL C01767 V=800.0 PL=0
MOVL C01768 V=800.0 PL=0
MOVL C01769 V=800.0 PL=0
MOVL C01770 V=800.0 PL=0
MOVL C01771 V=800.0 PL=0
MOVL C01772 V=800.0 PL=0
MOVL C01773 V=800.0 PL=0
MOVL C01774 V=800.0 PL=0
MOVL C01775 V=800.0 PL=0
MOVL C01776 V=800.0 PL=0
MOVL C01777 V=800.0 PL=0
MOVL C01778 V=800.0 PL=0
MOVL C01779 V=800.0 PL=0
MOVL C01780 V=800.0 PL=0
MOVL C01781 V=800.0 PL=0
MOVL C01782 V=800.0 PL=0
MOVL C01783 V=800.0 PL=0
MOVL C01784 V=800.0 PL=0
MOVL C01785 V=800.0 PL=0
MOVL C01786 V=800.0 PL=0
MOVL C01787 V=800.0 PL=0
MOVL C01788 V=800.0 PL=0
MOVL C01789 V=800.0 PL=0
MOVL C01790 V=800.0 PL=0
MOVL C01791 V=800.0 PL=0
MOVL C01792 V=800.0 PL=0
MOVL C01793 V=800.0 PL=0
MOVL C01794 V=800.0 PL=0
MOVL C01795 V=800.0 PL=0
MOVL C01796 V=800.0 PL=0
MOVL C01797 V=800.0 PL=0
MOVL C01798 V=800.0 PL=0
MOVL C01799 V=800.0 PL=0
MOVL C01800 V=800.0 PL=0
MOVL C01801 V=800.0 PL=0
MOVL C01802 V=800.0 PL=0
MOVL C01803 V=800.0 PL=0
MOVL C01804 V=800.0 PL=0
MOVL C01805 V=800.0 PL=0
MOVL C01806 V=800.0 PL=0
MOVL C01807 V=800.0 PL=0
MOVL C01808 V=800.0 PL=0
MOVL C01809 V=800.0 PL=0
MOVL C01810 V=800.0 PL=0
MOVL C01811 V=800.0 PL=0
MOVL C01812 V=800.0 PL=0
MOVL C01813 V=800.0 PL=0
MOVL C01814 V=800.0 PL=0
MOVL C01815 V=800.0 PL=0
MOVL C01816 V=800.0 PL=0
MOVL C01817 V=800.0 PL=0
MOVL C01818 V=800.0 PL=0
MOVL C01819 V=800.0 PL=0
MOVL C01820 V=800.0 PL=0
MOVL C01821 V=800.0 PL=0
MOVL C01822 V=800.0 PL=0
MOVL C01823 V=800.0 PL=0
MOVL C01824 V=800.0 PL=0
MOVL C01825 V=800.0 PL=0
MOVL C01826 V=800.0 PL=0
MOVL C01827 V=800.0 PL=0
MOVL C01828 V=800.0 PL=0
MOVL C01829 V=800.0 PL=0
MOVL C01830 V=800.0 PL=0
MOVL C01831 V=800.0 PL=0
MOVL C01832 V=800.0 PL=0
MOVL C01833 V=800.0 PL=0
MOVL C01834 V=800.0 PL=0
MOVL C01835 V=800.0 PL=0
MOVL C01836 V=800.0 PL=0
MOVL C01837 V=800.0 PL=0
MOVL C01838 V=800.0 PL=0
MOVL C01839 V=800.0 PL=0
MOVL C01840 V=800.0 PL=0
MOVL C01841 V=800.0 PL=0
MOVL C01842 V=800.0 PL=0
MOVL C01843 V=800.0 PL=0
MOVL C01844 V=800.0 PL=0
MOVL C01845 V=800.0 PL=0
MOVL C01846 V=800.0 PL=0
MOVL C01847 V=800.0 PL=0
MOVL C01848 V=800.0 PL=0
MOVL C01849 V=800.0 PL=0
MOVL C01850 V=800.0 PL=0
MOVL C01851 V=800.0 PL=0
MOVL C01852 V=800.0 PL=0
MOVL C01853 V=800.0 PL=0
MOVL C01854 V=800.0 PL=0
MOVL C01855 V=800.0 PL=0
MOVL C01856 V=800.0 PL=0
MOVL C01857 V=800.0 PL=0
MOVL C01858 V=800.0 PL=0
MOVL C01859 V=800.0 PL=0
MOVL C01860 V=800.0 PL=0
MOVL C01861 V=800.0 PL=0
MOVL C01862 V=800.0 PL=0
MOVL C01863 V=800.0 PL=0
MOVL C01864 V=800.0 PL=0
MOVL C01865 V=800.0 PL=0
MOVL C01866 V=800.0 PL=0
MOVL C01867 V=800.0 PL=0
MOVL C01868 V=800.0 PL=0
MOVL C01869 V=800.0 PL=0
MOVL C01870 V=800.0 PL=0
MOVL C01871 V=800.0 PL=0
MOVL C01872 V=800.0 PL=0
MOVL C01873 V=800.0 PL=0
MOVL C01874 V=800.0 PL=0
MOVL C01875 V=800.0 PL=0
MOVL C01876 V=800.0 PL=0
MOVL C01877 V=800.0 PL=0
MOVL C01878 V=800.0 PL=0
MOVL C01879 V=800.0 PL=0
MOVL C01880 V=800.0 PL=0
MOVL C01881 V=800.0 PL=0
MOVL C01882 V=800.0 PL=0
MOVL C01883 V=800.0 PL=0
MOVL C01884 V=800.0 PL=0
MOVL C01885 V=800.0 PL=0
MOVL C01886 V=800.0 PL=0
MOVL C01887 V=800.0 PL=0
MOVL C01888 V=800.0 PL=0
MOVL C01889 V=800.0 PL=0
MOVL C01890 V=800.0 PL=0
MOVL C01891 V=800.0 PL=0
MOVL C01892 V=800.0 PL=0
MOVL C01893 V=800.0 PL=0
MOVL C01894 V=800.0 PL=0
MOVL C01895 V=800.0 PL=0
MOVL C01896 V=800.0 PL=0
MOVL C01897 V=800.0 PL=0
MOVL C01898 V=800.0 PL=0
MOVL C01899 V=800.0 PL=0
MOVL C01900 V=800.0 PL=0
MOVL C01901 V=800.0 PL=0
MOVL C01902 V=800.0 PL=0
MOVL C01903 V=800.0 PL=0
MOVL C01904 V=800.0 PL=0
MOVL C01905 V=800.0 PL=0
MOVL C01906 V=800.0 PL=0
MOVL C01907 V=800.0 PL=0
MOVL C01908 V=800.0 PL=0
MOVL C01909 V=800.0 PL=0
MOVL C01910 V=800.0 PL=0
MOVL C01911 V=800.0 PL=0
MOVL C01912 V=800.0 PL=0
MOVL C01913 V=800.0 PL=0
MOVL C01914 V=800.0 PL=0
MOVL C01915 V=800.0 PL=0
MOVL C01916 V=800.0 PL=0
MOVL C01917 V=800.0 PL=0
MOVL C01918 V=800.0 PL=0
MOVL C01919 V=800.0 PL=0
MOVL C01920 V=800.0 PL=0
MOVL C01921 V=800.0 PL=0
MOVL C01922 V=800.0 PL=0
MOVL C01923 V=800.0 PL=0
MOVL C01924 V=800.0 PL=0
MOVL C01925 V=800.0 PL=0
MOVL C01926 V=800.0 PL=0
MOVL C01927 V=800.0 PL=0
MOVL C01928 V=800.0 PL=0
MOVL C01929 V=800.0 PL=0
MOVL C01930 V=800.0 PL=0
MOVL C01931 V=800.0 PL=0
MOVL C01932 V=800.0 PL=0
MOVL C01933 V=800.0 PL=0
MOVL C01934 V=800.0 PL=0
MOVL C01935 V=800.0 PL=0
MOVL C01936 V=800.0 PL=0
MOVL C01937 V=800.0 PL=0
MOVL C01938 V=800.0 PL=0
MOVL C01939 V=800.0 PL=0
MOVL C01940 V=800.0 PL=0
MOVL C01941 V=800.0 PL=0
MOVL C01942 V=800.0 PL=0
MOVL C01943 V=800.0 PL=0
MOVL C01944 V=800.0 PL=0
MOVL C01945 V=800.0 PL=0
MOVL C01946 V=800.0 PL=0
MOVL C01947 V=800.0 PL=0
MOVL C01948 V=800.0 PL=0
MOVL C01949 V=800.0 PL=0
MOVL C01950 V=800.0 PL=0
MOVL C01951 V=800.0 PL=0
MOVL C01952 V=800.0 PL=0
